KUKA KRL program: MyProgram_066().src

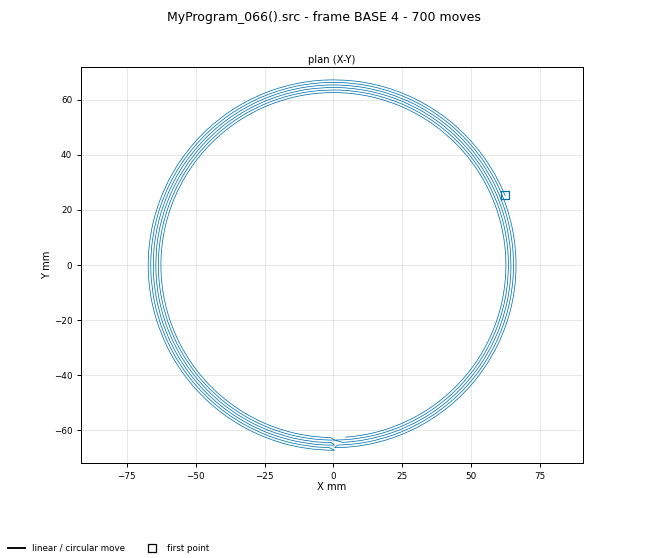
[picture p0: tool path of MyProgram_066().src in frame BASE 4, 700 of 700 moves have a stored position in this frame; points joined in program order, loops and branches not executed]
&ACCESS RVP
&REL 1
&PARAM TEMPLATE = C:\KRC\Roboter\Template\vorgabe
&PARAM EDITMASK = *
DEF MyProgram_066()
; ---- Setting reference (Base) ----
$BASE = BASE_DATA[4]

; --------------------------
; ---- Setting tool (TCP) ----
$TOOL = TOOL_DATA[3]
; --------------------------

$VEL.CP = VEL_APROX_PRINT
Startdeposition()
$VEL.CP = VEL_PRINT
LIN {X 62.3315,Y 25.2881,Z 74,A 16.8534,B 24.8789,C -2.5402,E1 25.1473,E2 67.2399} C_DIS
LIN {X 60.7324,Y 28.9196,Z 74,A 20.0242,B 24.8785,C -2.5441,E1 25.1436,E2 64.0772} C_DIS
LIN {X 58.523,Y 33.1652,Z 74,A 24.2572,B 24.877,C -2.5592,E1 25.138,E2 59.8308} C_DIS
LIN {X 56.2659,Y 36.8633,Z 74,A 27.5694,B 24.877,C -2.5587,E1 25.1331,E2 56.5365} C_DIS
LIN {X 55.2782,Y 38.328,Z 74,A 29.4981,B 24.8757,C -2.5736,E1 25.13,E2 54.5819} C_DIS
LIN {X 52.9232,Y 41.5199,Z 74,A 32.7172,B 24.8753,C -2.5775,E1 25.1246,E2 51.369} C_DIS
LIN {X 49.6306,Y 45.404,Z 74,A 36.4526,B 24.8758,C -2.5716,E1 25.1179,E2 47.6643} C_DIS
LIN {X 47.2788,Y 47.848,Z 74,A 39.6344,B 24.8745,C -2.5853,E1 25.1116,E2 44.4638} C_DIS
LIN {X 44.4374,Y 50.4985,Z 74,A 42.7954,B 24.8742,C -2.5881,E1 25.1051,E2 41.309} C_DIS
LIN {X 41.8737,Y 52.6437,Z 74,A 45.7271,B 24.8735,C -2.5955,E1 25.0988,E2 38.371} C_DIS
LIN {X 38.9575,Y 54.8366,Z 74,A 49.1887,B 24.8721,C -2.6099,E1 25.091,E2 34.8877} C_DIS
LIN {X 35.2683,Y 57.2802,Z 74,A 52.5369,B 24.8726,C -2.6051,E1 25.0832,E2 31.5619} C_DIS
LIN {X 32.0783,Y 59.1244,Z 74,A 55.3853,B 24.8729,C -2.6022,E1 25.0763,E2 28.7288} C_DIS
LIN {X 29.6751,Y 60.3668,Z 74,A 58.2734,B 24.8712,C -2.6196,E1 25.0691,E2 25.8073} C_DIS
LIN {X 27.6413,Y 61.3243,Z 74,A 60.3296,B 24.8706,C -2.6253,E1 25.0638,E2 23.7428} C_DIS
LIN {X 24.27,Y 62.736,Z 74,A 63.3703,B 24.8705,C -2.6266,E1 25.0559,E2 20.7059} C_DIS
LIN {X 20.9505,Y 63.9207,Z 74,A 66.4008,B 24.8701,C -2.6298,E1 25.0479,E2 17.6737} C_DIS
LIN {X 17.9241,Y 64.8352,Z 74,A 69.0945,B 24.87,C -2.6317,E1 25.0407,E2 14.9802} C_DIS
LIN {X 13.9191,Y 65.8114,Z 74,A 72.377,B 24.8703,C -2.6279,E1 25.0318,E2 11.7111} C_DIS
LIN {X 10.864,Y 66.3823,Z 74,A 75.0856,B 24.8701,C -2.6304,E1 25.0243,E2 8.9996} C_DIS
LIN {X 7.712,Y 66.8226,Z 74,A 77.9948,B 24.8696,C -2.6357,E1 25.0163,E2 6.0801} C_DIS
LIN {X 4.131,Y 67.1403,Z 74,A 80.6016,B 24.8706,C -2.625,E1 25.0091,E2 3.5} C_DIS
LIN {X -0.3651,Y 67.265,Z 74,A 84.501,B 24.8706,C -2.6261,E1 24.9982,E2 -0.4014} C_DIS
LIN {X -3.8279,Y 67.1571,Z 74,A 88.2033,B 24.8689,C -2.6427,E1 24.9877,E2 -4.1439} C_DIS
LIN {X -7.4514,Y 66.8531,Z 74,A 90.84,B 24.8701,C -2.6303,E1 24.9805,E2 -6.7528} C_DIS
LIN {X -10.4471,Y 66.45,Z 74,A 93.2751,B 24.8706,C -2.6255,E1 24.9738,E2 -9.1784} C_DIS
LIN {X -12.9697,Y 66.0043,Z 74,A 95.4752,B 24.8706,C -2.6242,E1 24.9678,E2 -11.3777} C_DIS
LIN {X -16.4947,Y 65.2128,Z 74,A 99.486,B 24.8689,C -2.6426,E1 24.9567,E2 -15.438} C_DIS
LIN {X -19.9918,Y 64.2265,Z 74,A 101.0557,B 24.8726,C -2.6048,E1 24.9528,E2 -16.9203} C_DIS
LIN {X -23.3556,Y 63.082,Z 74,A 104.7013,B 24.8716,C -2.6149,E1 24.9431,E2 -20.5968} C_DIS
LIN {X -25.7788,Y 62.1314,Z 74,A 107.2724,B 24.8711,C -2.6197,E1 24.9364,E2 -23.1852} C_DIS
LIN {X -29.9946,Y 60.2084,Z 74,A 110.6168,B 24.873,C -2.6004,E1 24.928,E2 -26.492} C_DIS
LIN {X -31.8168,Y 59.2655,Z 74,A 112.8643,B 24.8722,C -2.6085,E1 24.9224,E2 -28.765} C_DIS
LIN {X -35.093,Y 57.3867,Z 74,A 115.6735,B 24.8737,C -2.5939,E1 24.9157,E2 -31.5478} C_DIS
LIN {X -36.6852,Y 56.3816,Z 74,A 117.6551,B 24.8732,C -2.5991,E1 24.911,E2 -33.5482} C_DIS
LIN {X -39.5297,Y 54.426,Z 74,A 120.8352,B 24.8732,C -2.5984,E1 24.9038,E2 -36.7377} C_DIS
LIN {X -43.4881,Y 51.318,Z 74,A 124.3334,B 24.8758,C -2.5723,E1 24.8963,E2 -40.1869} C_DIS
LIN {X -45.912,Y 49.1611,Z 74,A 127.8706,B 24.8748,C -2.5825,E1 24.8889,E2 -43.7626} C_DIS
LIN {X -49.0981,Y 45.9794,Z 74,A 131.8946,B 24.8753,C -2.5773,E1 24.8811,E2 -47.7914} C_DIS
LIN {X -51.4905,Y 43.285,Z 74,A 134.9532,B 24.8761,C -2.5693,E1 24.8755,E2 -50.8448} C_DIS
LIN {X -54.426,Y 39.5297,Z 74,A 138.5981,B 24.878,C -2.5498,E1 24.8694,E2 -54.4606} C_DIS
LIN {X -56.1384,Y 37.0567,Z 74,A 141.0375,B 24.8789,C -2.5402,E1 24.8656,E2 -56.8894} C_DIS
LIN {X -57.3949,Y 35.0794,Z 74,A 143.5728,B 24.8783,C -2.5459,E1 24.8619,E2 -59.4512} C_DIS
LIN {X -59.9905,Y 30.4285,Z 74,A 148.1441,B 24.8795,C -2.5336,E1 24.8559,E2 -64.0172} C_DIS
LIN {X -62.1829,Y 25.6534,Z 74,A 152.2818,B 24.8814,C -2.5132,E1 24.8512,E2 -68.129} C_DIS
LIN {X -63.6586,Y 21.734,Z 74,A 155.9508,B 24.8823,C -2.5044,E1 24.8477,E2 -71.7979} C_DIS
LIN {X -64.7804,Y 18.1175,Z 74,A 159.2016,B 24.8832,C -2.495,E1 24.8452,E2 -75.0449} C_DIS
LIN {X -65.5151,Y 15.2482,Z 74,A 161.5576,B 24.8842,C -2.4837,E1 24.8436,E2 -77.3876} C_DIS
LIN {X -65.9957,Y 13.0146,Z 74,A 163.4166,B 24.885,C -2.4758,E1 24.8426,E2 -79.2387} C_DIS
LIN {X -66.7571,Y 8.2673,Z 74,A 167.478,B 24.8862,C -2.4621,E1 24.8409,E2 -83.2917} C_DIS
LIN {X -67.1045,Y 4.6607,Z 74,A 171.2927,B 24.8857,C -2.4673,E1 24.84,E2 -87.1417} C_DIS
LIN {X -67.2573,Y 1.0908,Z 74,A 174.6764,B 24.886,C -2.4648,E1 24.8398,E2 -90.5396} C_DIS
LIN {X -67.2266,Y -2.3165,Z 74,A 176.844,B 24.8882,C -2.4404,E1 24.84,E2 -92.662} C_DIS
LIN {X -67.0976,Y -4.7627,Z 74,A 179.1127,B 24.8885,C -2.4376,E1 24.8404,E2 -94.9376} C_DIS
LIN {X -66.7559,Y -8.277,Z 74,A -177.9869,B 24.8895,C -2.426,E1 24.8413,E2 -97.8276} C_DIS
LIN {X -66.2127,Y -11.8575,Z 74,A -174.9721,B 24.8905,C -2.415,E1 24.8426,E2 -100.8342} C_DIS
LIN {X -65.7862,Y -14.0352,Z 74,A -172.2602,B 24.8895,C -2.4264,E1 24.8442,E2 -103.5892} C_DIS
LIN {X -65.0081,Y -17.2788,Z 74,A -170.101,B 24.8916,C -2.4036,E1 24.8457,E2 -105.7065} C_DIS
LIN {X -64.2056,Y -20.0594,Z 74,A -167.7944,B 24.8925,C -2.3929,E1 24.8476,E2 -108.001} C_DIS
LIN {X -63.5273,Y -22.114,Z 74,A -165.4328,B 24.8921,C -2.3984,E1 24.8497,E2 -110.3891} C_DIS
LIN {X -61.4519,Y -27.3582,Z 74,A -161.3561,B 24.8946,C -2.3695,E1 24.854,E2 -114.4193} C_DIS
LIN {X -60.244,Y -29.923,Z 74,A -158.4157,B 24.8943,C -2.3738,E1 24.8576,E2 -117.3862} C_DIS
LIN {X -58.7607,Y -32.7395,Z 74,A -155.6768,B 24.8949,C -2.3672,E1 24.8613,E2 -120.1237} C_DIS
LIN {X -57.5024,Y -34.9027,Z 74,A -153.0961,B 24.8945,C -2.3712,E1 24.865,E2 -122.7273} C_DIS
LIN {X -55.1447,Y -38.5202,Z 74,A -150.0261,B 24.8965,C -2.349,E1 24.8698,E2 -125.7595} C_DIS
LIN {X -53.5092,Y -40.763,Z 74,A -147.4333,B 24.8965,C -2.3482,E1 24.8741,E2 -128.3628} C_DIS
LIN {X -51.3233,Y -43.4818,Z 74,A -144.7496,B 24.8977,C -2.3352,E1 24.8789,E2 -131.0278} C_DIS
LIN {X -49.4277,Y -45.6252,Z 74,A -142.4389,B 24.8984,C -2.3271,E1 24.8832,E2 -133.3295} C_DIS
LIN {X -47.0995,Y -48.0251,Z 74,A -139.4796,B 24.8987,C -2.3235,E1 24.889,E2 -136.293} C_DIS
LIN {X -45.2438,Y -49.7777,Z 74,A -137.0243,B 24.8985,C -2.3253,E1 24.894,E2 -138.7626} C_DIS
LIN {X -43.3659,Y -51.4221,Z 74,A -134.2375,B 24.8976,C -2.336,E1 24.9001,E2 -141.5856} C_DIS
LIN {X -40.7193,Y -53.5426,Z 74,A -131.2988,B 24.898,C -2.3321,E1 24.9066,E2 -144.5256} C_DIS
LIN {X -37.9226,Y -55.5577,Z 74,A -129.4698,B 24.9005,C -2.3026,E1 24.9107,E2 -146.2904} C_DIS
LIN {X -34.8215,Y -57.5517,Z 74,A -125.8623,B 24.9,C -2.3083,E1 24.9192,E2 -149.923} C_DIS
LIN {X -31.8372,Y -59.2552,Z 74,A -123.1085,B 24.9007,C -2.3005,E1 24.9259,E2 -152.6661} C_DIS
LIN {X -29.2171,Y -60.5895,Z 74,A -120.3691,B 24.9005,C -2.3028,E1 24.9328,E2 -155.4183} C_DIS
LIN {X -25.5883,Y -62.2094,Z 74,A -117.097,B 24.901,C -2.2967,E1 24.9412,E2 -158.6834} C_DIS
LIN {X -21.9524,Y -63.5838,Z 74,A -113.698,B 24.9011,C -2.2959,E1 24.9501,E2 -162.0873} C_DIS
LIN {X -18.3294,Y -64.7205,Z 74,A -110.5135,B 24.9014,C -2.2925,E1 24.9586,E2 -165.2691} C_DIS
LIN {X -16.0949,Y -65.3123,Z 74,A -107.5998,B 24.8995,C -2.3138,E1 24.9667,E2 -168.2377} C_DIS
LIN {X -12.1273,Y -66.1641,Z 74,A -103.8828,B 24.8991,C -2.3189,E1 24.977,E2 -171.9705} C_DIS
LIN {X -7.472,Y -66.8507,Z 74,A -100.7261,B 24.901,C -2.2977,E1 24.9856,E2 -175.0788} C_DIS
LIN {X -2.0633,Y -67.2344,Z 74,A -96.425,B 24.9016,C -2.2902,E1 24.9975,E2 -179.3634} C_DIS
LIN {X 0.449,Y -67.2547,Z 74,A -94.5441,B 24.9021,C -2.2846,E1 25.0027,E2 -181.2309} C_DIS
Enddeposition()
LIN {X 0.449,Y -67.2547,Z 74,A -94.5441,B 24.9021,C -2.2846,E1 25.0027,E2 -181.2309} C_DIS
Startdeposition()
$VEL.CP = VEL_PRINT
LIN {X -1.4149,Y -66.3279,Z 74,A -97.2166,B 24.9029,C -2.2748,E1 24.9952,E2 -178.5352} C_DIS
LIN {X -6.4726,Y -66.0273,Z 74,A -101.5733,B 24.9029,C -2.2752,E1 24.9831,E2 -174.1777} C_DIS
LIN {X -11.6127,Y -65.3185,Z 74,A -105.8847,B 24.9025,C -2.2802,E1 24.9712,E2 -169.8746} C_DIS
LIN {X -14.9653,Y -64.6327,Z 74,A -108.7487,B 24.9022,C -2.2835,E1 24.9634,E2 -167.015} C_DIS
LIN {X -17.1256,Y -64.0944,Z 74,A -111.8991,B 24.9044,C -2.2571,E1 24.9547,E2 -163.7972} C_DIS
LIN {X -20.6683,Y -63.0415,Z 74,A -114.2557,B 24.9026,C -2.278,E1 24.9486,E2 -161.486} C_DIS
LIN {X -22.9852,Y -62.2343,Z 74,A -116.4421,B 24.9026,C -2.2783,E1 24.9428,E2 -159.296} C_DIS
LIN {X -25.3695,Y -61.3016,Z 74,A -118.9919,B 24.9031,C -2.2731,E1 24.9362,E2 -156.728} C_DIS
LIN {X -30.5306,Y -58.9014,Z 74,A -123.945,B 24.9026,C -2.2781,E1 24.9237,E2 -151.774} C_DIS
LIN {X -34.4147,Y -56.7185,Z 74,A -127.7165,B 24.902,C -2.2852,E1 24.9147,E2 -148.008} C_DIS
LIN {X -37.3127,Y -54.8555,Z 74,A -130.8798,B 24.902,C -2.2859,E1 24.9073,E2 -144.8358} C_DIS
LIN {X -40.1239,Y -52.835,Z 74,A -133.2241,B 24.9003,C -2.3047,E1 24.9021,E2 -142.528} C_DIS
LIN {X -42.9208,Y -50.5883,Z 74,A -136.3928,B 24.9,C -2.3089,E1 24.8953,E2 -139.3573} C_DIS
LIN {X -45.6353,Y -48.1543,Z 74,A -139.6748,B 24.8997,C -2.3123,E1 24.8885,E2 -136.0701} C_DIS
LIN {X -48.3948,Y -45.3796,Z 74,A -143.0463,B 24.899,C -2.3196,E1 24.882,E2 -132.7017} C_DIS
LIN {X -50.6642,Y -42.8317,Z 74,A -146.3244,B 24.899,C -2.3194,E1 24.876,E2 -129.4082} C_DIS
LIN {X -52.8948,Y -40.0444,Z 74,A -148.636,B 24.897,C -2.3426,E1 24.8721,E2 -127.1409} C_DIS
LIN {X -54.1488,Y -38.3318,Z 74,A -151.1998,B 24.898,C -2.332,E1 24.8678,E2 -124.5394} C_DIS
LIN {X -56.7395,Y -34.38,Z 74,A -154.6858,B 24.896,C -2.3546,E1 24.8626,E2 -121.0896} C_DIS
LIN {X -57.9531,Y -32.2924,Z 74,A -156.8887,B 24.8957,C -2.3577,E1 24.8596,E2 -118.8827} C_DIS
LIN {X -59.2868,Y -29.7714,Z 74,A -159.8608,B 24.896,C -2.3541,E1 24.8557,E2 -115.8861} C_DIS
LIN {X -61.0479,Y -25.9716,Z 74,A -163.5382,B 24.8952,C -2.363,E1 24.8516,E2 -112.2098} C_DIS
LIN {X -62.6169,Y -21.9197,Z 74,A -167.4766,B 24.8946,C -2.3702,E1 24.8478,E2 -108.2663} C_DIS
LIN {X -64.2281,Y -16.6168,Z 74,A -172.1789,B 24.8932,C -2.3862,E1 24.8442,E2 -103.5749} C_DIS
LIN {X -64.8986,Y -13.7717,Z 74,A -174.371,B 24.8919,C -2.4004,E1 24.8429,E2 -101.4039} C_DIS
LIN {X -65.4441,Y -10.8822,Z 74,A -177.4683,B 24.8922,C -2.3972,E1 24.8414,E2 -98.2807} C_DIS
LIN {X -66.1466,Y -5.0997,Z 74,A 178.2949,B 24.8893,C -2.4286,E1 24.8402,E2 -94.0934} C_DIS
LIN {X -66.2816,Y -2.8454,Z 74,A 176.1064,B 24.8892,C -2.43,E1 24.8399,E2 -91.8952} C_DIS
LIN {X -66.3414,Y 0.3365,Z 74,A 173.5212,B 24.8881,C -2.4419,E1 24.8398,E2 -89.3229} C_DIS
LIN {X -66.3053,Y 2.2349,Z 74,A 171.3771,B 24.8885,C -2.4372,E1 24.84,E2 -87.1546} C_DIS
LIN {X -66.0051,Y 6.6877,Z 74,A 167.8104,B 24.8869,C -2.455,E1 24.8408,E2 -83.6091} C_DIS
LIN {X -65.6576,Y 9.5109,Z 74,A 164.9106,B 24.8869,C -2.4541,E1 24.8419,E2 -80.6897} C_DIS
LIN {X -65.0311,Y 13.1272,Z 74,A 162.0301,B 24.8855,C -2.4698,E1 24.8434,E2 -77.8296} C_DIS
LIN {X -64.3433,Y 16.1686,Z 74,A 159.3509,B 24.8847,C -2.4784,E1 24.8451,E2 -75.1554} C_DIS
LIN {X -63.4775,Y 19.2866,Z 74,A 156.7155,B 24.8836,C -2.4902,E1 24.8471,E2 -72.5329} C_DIS
LIN {X -62.1556,Y 23.1965,Z 74,A 152.8909,B 24.8831,C -2.496,E1 24.8507,E2 -68.7003} C_DIS
LIN {X -60.5332,Y 27.1485,Z 74,A 148.6944,B 24.883,C -2.497,E1 24.8553,E2 -64.4832} C_DIS
LIN {X -58.8514,Y 30.625,Z 74,A 145.5471,B 24.8817,C -2.5104,E1 24.8593,E2 -61.351} C_DIS
LIN {X -56.7052,Y 34.4365,Z 74,A 142.0487,B 24.8802,C -2.5267,E1 24.8641,E2 -57.8732} C_DIS
LIN {X -54.8734,Y 37.2862,Z 74,A 139.3938,B 24.8789,C -2.5401,E1 24.8682,E2 -55.2372} C_DIS
LIN {X -53.7459,Y 38.8956,Z 74,A 137.4149,B 24.8789,C -2.539,E1 24.8714,E2 -53.246} C_DIS
LIN {X -51.8231,Y 41.4228,Z 74,A 134.5691,B 24.8785,C -2.5441,E1 24.8763,E2 -50.3989} C_DIS
LIN {X -49.4365,Y 44.2423,Z 74,A 131.2964,B 24.8779,C -2.5505,E1 24.8823,E2 -47.1266} C_DIS
LIN {X -46.9076,Y 46.9168,Z 74,A 128.1251,B 24.8771,C -2.5583,E1 24.8885,E2 -43.9602} C_DIS
LIN {X -44.1214,Y 49.5442,Z 74,A 125.2179,B 24.8756,C -2.5741,E1 24.8944,E2 -41.0789} C_DIS
LIN {X -41.71,Y 51.5909,Z 74,A 122.0987,B 24.8758,C -2.572,E1 24.9011,E2 -37.9429} C_DIS
LIN {X -38.912,Y 53.7338,Z 74,A 119.2437,B 24.8748,C -2.5821,E1 24.9075,E2 -35.1018} C_DIS
LIN {X -36.9584,Y 55.0946,Z 74,A 117.076,B 24.8747,C -2.5838,E1 24.9125,E2 -32.9309} C_DIS
LIN {X -34.4679,Y 56.6861,Z 74,A 114.2062,B 24.8748,C -2.5819,E1 24.9193,E2 -30.0475} C_DIS
LIN {X -30.1508,Y 59.0955,Z 74,A 110.3017,B 24.8734,C -2.5967,E1 24.9288,E2 -26.1673} C_DIS
LIN {X -27.0922,Y 60.559,Z 74,A 106.9855,B 24.8738,C -2.5929,E1 24.9373,E2 -22.8338} C_DIS
LIN {X -23.5832,Y 62.0096,Z 74,A 103.7025,B 24.8734,C -2.5972,E1 24.9458,E2 -19.5539} C_DIS
LIN {X -20.5647,Y 63.0751,Z 74,A 101.4564,B 24.8719,C -2.6117,E1 24.9517,E2 -17.3381} C_DIS
LIN {X -16.4891,Y 64.2609,Z 74,A 97.9439,B 24.8712,C -2.6189,E1 24.9611,E2 -13.8371} C_DIS
LIN {X -13.3428,Y 64.9871,Z 74,A 95.0047,B 24.8713,C -2.6181,E1 24.9691,E2 -10.8921} C_DIS
LIN {X -11.5671,Y 65.3268,Z 74,A 93.1162,B 24.8719,C -2.612,E1 24.9743,E2 -8.9872} C_DIS
LIN {X -7.9595,Y 65.8639,Z 74,A 90.3042,B 24.871,C -2.6215,E1 24.982,E2 -6.1956} C_DIS
LIN {X -4.1713,Y 66.2121,Z 74,A 86.3277,B 24.8723,C -2.6075,E1 24.9932,E2 -2.1841} C_DIS
LIN {X -0.5098,Y 66.3408,Z 74,A 82.8327,B 24.873,C -2.6009,E1 25.003,E2 1.3268} C_DIS
LIN {X 2.8294,Y 66.2823,Z 74,A 81.3016,B 24.8699,C -2.6319,E1 25.0071,E2 2.7839} C_DIS
LIN {X 4.7605,Y 66.1723,Z 74,A 78.5897,B 24.8723,C -2.608,E1 25.0148,E2 5.5513} C_DIS
LIN {X 9.6031,Y 65.6446,Z 74,A 74.5516,B 24.872,C -2.611,E1 25.0259,E2 9.5791} C_DIS
LIN {X 12.7089,Y 65.1142,Z 74,A 72.1013,B 24.8715,C -2.6162,E1 25.0326,E2 12.0142} C_DIS
LIN {X 16.0999,Y 64.3597,Z 74,A 69.1183,B 24.8716,C -2.6151,E1 25.0407,E2 14.9958} C_DIS
LIN {X 20.0962,Y 63.2267,Z 74,A 65.8599,B 24.8711,C -2.6203,E1 25.0494,E2 18.2362} C_DIS
LIN {X 24.5864,Y 61.6194,Z 74,A 61.0061,B 24.8732,C -2.5991,E1 25.0622,E2 23.1301} C_DIS
LIN {X 27.6395,Y 60.3122,Z 74,A 58.4966,B 24.8726,C -2.6045,E1 25.0686,E2 25.6207} C_DIS
LIN {X 31.5817,Y 58.3434,Z 74,A 54.322,B 24.874,C -2.5907,E1 25.079,E2 29.8162} C_DIS
LIN {X 34.8131,Y 56.4761,Z 74,A 50.7144,B 24.8754,C -2.5767,E1 25.0876,E2 33.4458} C_DIS
LIN {X 37.7449,Y 54.5591,Z 74,A 47.7125,B 24.8758,C -2.5723,E1 25.0945,E2 36.4478} C_DIS
LIN {X 40.5739,Y 52.4893,Z 74,A 46.1787,B 24.8727,C -2.6038,E1 25.0978,E2 37.9015} C_DIS
LIN {X 42.6402,Y 50.8257,Z 74,A 43.3374,B 24.8745,C -2.5859,E1 25.104,E2 40.7745} C_DIS
LIN {X 44.2021,Y 49.4725,Z 74,A 41.099,B 24.8759,C -2.5711,E1 25.1087,E2 43.0389} C_DIS
LIN {X 46.5542,Y 47.2659,Z 74,A 38.3066,B 24.8765,C -2.5652,E1 25.1143,E2 45.8337} C_DIS
LIN {X 48.7959,Y 44.9481,Z 74,A 36.1102,B 24.8756,C -2.5739,E1 25.1185,E2 47.9998} C_DIS
LIN {X 51.1276,Y 42.2771,Z 74,A 32.8841,B 24.8767,C -2.5628,E1 25.1244,E2 51.2377} C_DIS
LIN {X 53.4624,Y 39.2827,Z 74,A 29.9082,B 24.8767,C -2.5627,E1 25.1294,E2 54.1996} C_DIS
LIN {X 54.7371,Y 37.4876,Z 74,A 27.6827,B 24.878,C -2.5497,E1 25.133,E2 56.445} C_DIS
LIN {X 57.5072,Y 33.0798,Z 74,A 23.595,B 24.878,C -2.5486,E1 25.139,E2 60.5147} C_DIS
LIN {X 59.3392,Y 29.6693,Z 74,A 20.1707,B 24.8791,C -2.5374,E1 25.1434,E2 63.9472} C_DIS
LIN {X 60.8589,Y 26.4102,Z 74,A 16.1566,B 24.8822,C -2.5053,E1 25.1481,E2 68.0154} C_DIS
LIN {X 62.4219,Y 22.4707,Z 74,A 12.8782,B 24.8822,C -2.5045,E1 25.1513,E2 71.2773} C_DIS
LIN {X 63.5424,Y 19.0726,Z 74,A 9.9293,B 24.8828,C -2.4991,E1 25.1537,E2 74.2224} C_DIS
LIN {X 64.6929,Y 14.705,Z 74,A 6.7032,B 24.8822,C -2.5049,E1 25.1559,E2 77.416} C_DIS
LIN {X 65.4196,Y 11.0285,Z 74,A 3.1661,B 24.8839,C -2.4871,E1 25.1578,E2 80.9747} C_DIS
LIN {X 65.9012,Y 7.6411,Z 74,A -0.297,B 24.886,C -2.4646,E1 25.159,E2 84.4705} C_DIS
LIN {X 66.3011,Y 2.3596,Z 74,A -5.0224,B 24.8877,C -2.4462,E1 25.1598,E2 89.2111} C_DIS
LIN {X 66.3122,Y -2.0111,Z 74,A -8.7803,B 24.8887,C -2.4347,E1 25.1596,E2 92.9739} C_DIS
LIN {X 66.1167,Y -5.4741,Z 74,A -11.2155,B 24.8883,C -2.4399,E1 25.1591,E2 95.3824} C_DIS
LIN {X 65.8624,Y -7.9729,Z 74,A -14.1349,B 24.8907,C -2.4134,E1 25.1581,E2 98.3473} C_DIS
LIN {X 65.3481,Y -11.4482,Z 74,A -16.3481,B 24.8896,C -2.4252,E1 25.1571,E2 100.5194} C_DIS
LIN {X 64.6009,Y -15.103,Z 74,A -19.0559,B 24.8893,C -2.4287,E1 25.1555,E2 103.2033} C_DIS
LIN {X 63.9973,Y -17.485,Z 74,A -21.728,B 24.8912,C -2.4075,E1 25.1536,E2 105.91} C_DIS
LIN {X 62.9902,Y -20.8263,Z 74,A -24.4104,B 24.8912,C -2.4069,E1 25.1514,E2 108.5786} C_DIS
LIN {X 62.405,Y -22.517,Z 74,A -26.3509,B 24.8926,C -2.3918,E1 25.1495,E2 110.5438} C_DIS
LIN {X 61.0444,Y -25.9805,Z 74,A -29.3909,B 24.8931,C -2.3867,E1 25.1463,E2 113.5793} C_DIS
LIN {X 59.7124,Y -28.9106,Z 74,A -31.9702,B 24.8934,C -2.3837,E1 25.1433,E2 116.1516} C_DIS
LIN {X 58.693,Y -30.927,Z 74,A -34.428,B 24.8951,C -2.3648,E1 25.1401,E2 118.641} C_DIS
LIN {X 56.0131,Y -35.5528,Z 74,A -39.3479,B 24.8969,C -2.344,E1 25.1329,E2 123.5852} C_DIS
LIN {X 52.8789,Y -40.0655,Z 74,A -43.4784,B 24.8966,C -2.347,E1 25.1262,E2 127.6885} C_DIS
LIN {X 50.4209,Y -43.1173,Z 74,A -46.5566,B 24.8967,C -2.3462,E1 25.1208,E2 130.7545} C_DIS
LIN {X 48.7061,Y -45.0459,Z 74,A -49.3264,B 24.8984,C -2.3267,E1 25.1155,E2 133.558} C_DIS
LIN {X 45.8322,Y -47.9671,Z 74,A -52.5835,B 24.8985,C -2.3255,E1 25.109,E2 136.8045} C_DIS
LIN {X 42.9448,Y -50.5678,Z 74,A -55.619,B 24.8985,C -2.3261,E1 25.1027,E2 139.8264} C_DIS
LIN {X 40.8106,Y -52.3068,Z 74,A -58.6063,B 24.9003,C -2.3055,E1 25.0961,E2 142.8513} C_DIS
LIN {X 37.5193,Y -54.7157,Z 74,A -61.9311,B 24.9005,C -2.3034,E1 25.0885,E2 146.1696} C_DIS
LIN {X 33.7271,Y -57.13,Z 74,A -65.3568,B 24.9001,C -2.3076,E1 25.0805,E2 149.5743} C_DIS
LIN {X 30.4588,Y -58.9381,Z 74,A -69.1225,B 24.9017,C -2.2887,E1 25.0711,E2 153.3741} C_DIS
LIN {X 27.4535,Y -60.3962,Z 74,A -71.4428,B 24.9009,C -2.2982,E1 25.0653,E2 155.6661} C_DIS
LIN {X 24.8438,Y -61.5156,Z 74,A -74.1691,B 24.9018,C -2.2879,E1 25.0582,E2 158.4103} C_DIS
LIN {X 21.7194,Y -62.6872,Z 74,A -77.0242,B 24.9021,C -2.2848,E1 25.0507,E2 161.2668} C_DIS
LIN {X 19.056,Y -63.5473,Z 74,A -79.2329,B 24.9019,C -2.2871,E1 25.0449,E2 163.4661} C_DIS
LIN {X 15.7348,Y -64.4497,Z 74,A -82.1503,B 24.902,C -2.2854,E1 25.037,E2 166.383} C_DIS
LIN {X 13.1909,Y -65.0183,Z 74,A -85.667,B 24.9048,C -2.2532,E1 25.0272,E2 169.9716} C_DIS
LIN {X 9.0782,Y -65.7191,Z 74,A -88.0993,B 24.9026,C -2.2784,E1 25.0206,E2 172.3419} C_DIS
LIN {X 4.5562,Y -66.1861,Z 74,A -91.975,B 24.9026,C -2.2776,E1 25.0099,E2 176.2173} C_DIS
LIN {X 0.436,Y -66.3027,Z 74,A -94.6637,B 24.9009,C -2.2977,E1 25.0025,E2 178.8575} C_DIS
Enddeposition()
LIN {X 0.436,Y -66.3027,Z 74,A -94.6637,B 24.9009,C -2.2977,E1 25.0025,E2 178.8575} C_DIS
Startdeposition()
$VEL.CP = VEL_PRINT
LIN {X 1.5364,Y -65.4021,Z 74,A -92.9082,B 24.898,C -2.332,E1 25.0076,E2 177.021} C_DIS
LIN {X 6.6679,Y -65.0788,Z 74,A -88.8013,B 24.8986,C -2.3247,E1 25.019,E2 172.9336} C_DIS
LIN {X 9.6588,Y -64.7026,Z 74,A -85.5651,B 24.8972,C -2.3409,E1 25.028,E2 169.6618} C_DIS
LIN {X 13.0107,Y -64.1127,Z 74,A -83.4329,B 24.8988,C -2.3227,E1 25.0338,E2 167.5753} C_DIS
LIN {X 15.2589,Y -63.6154,Z 74,A -81.1168,B 24.898,C -2.3319,E1 25.0401,E2 165.2406} C_DIS
LIN {X 18.93,Y -62.6209,Z 74,A -78.0568,B 24.8982,C -2.3289,E1 25.0483,E2 162.1929} C_DIS
LIN {X 21.4935,Y -61.7879,Z 74,A -75.8242,B 24.8982,C -2.3287,E1 25.0542,E2 159.9653} C_DIS
LIN {X 24.6283,Y -60.6064,Z 74,A -72.403,B 24.8968,C -2.3448,E1 25.0631,E2 156.5135} C_DIS
LIN {X 27.6955,Y -59.2677,Z 74,A -69.3685,B 24.8962,C -2.3519,E1 25.0709,E2 153.4699} C_DIS
LIN {X 32.5774,Y -56.731,Z 74,A -65.2367,B 24.897,C -2.3428,E1 25.0809,E2 149.3714} C_DIS
LIN {X 37.0028,Y -53.9503,Z 74,A -60.1787,B 24.8952,C -2.3636,E1 25.0929,E2 144.2806} C_DIS
LIN {X 40.9187,Y -51.0438,Z 74,A -56.3828,B 24.8955,C -2.3604,E1 25.1013,E2 140.506} C_DIS
LIN {X 43.7208,Y -48.6627,Z 74,A -52.8437,B 24.8941,C -2.3759,E1 25.1088,E2 136.9443} C_DIS
LIN {X 46.6882,Y -45.8246,Z 74,A -48.9761,B 24.8927,C -2.3915,E1 25.1165,E2 133.0561} C_DIS
LIN {X 49.3002,Y -43.0021,Z 74,A -45.7073,B 24.8921,C -2.3974,E1 25.1225,E2 129.788} C_DIS
LIN {X 52.2689,Y -39.3403,Z 74,A -42.2274,B 24.8927,C -2.3913,E1 25.1285,E2 126.3388} C_DIS
LIN {X 54.8518,Y -35.6526,Z 74,A -38.1206,B 24.8913,C -2.4063,E1 25.135,E2 122.2167} C_DIS
LIN {X 56.3517,Y -33.2292,Z 74,A -35.5259,B 24.8905,C -2.416,E1 25.1388,E2 119.6124} C_DIS
LIN {X 57.9792,Y -30.3009,Z 74,A -32.7385,B 24.89,C -2.4206,E1 25.1425,E2 116.8287} C_DIS
LIN {X 59.5125,Y -27.167,Z 74,A -29.4159,B 24.8886,C -2.4366,E1 25.1464,E2 113.4861} C_DIS
LIN {X 60.8339,Y -24.0614,Z 74,A -26.7442,B 24.8884,C -2.4381,E1 25.1493,E2 110.8258} C_DIS
LIN {X 61.7874,Y -21.4951,Z 74,A -24.3517,B 24.8878,C -2.4452,E1 25.1515,E2 108.4297} C_DIS
LIN {X 62.6656,Y -18.7809,Z 74,A -21.1293,B 24.8853,C -2.4722,E1 25.1542,E2 105.1619} C_DIS
LIN {X 63.5166,Y -15.6641,Z 74,A -19.0424,B 24.8863,C -2.4613,E1 25.1556,E2 103.1129} C_DIS
LIN {X 64.4274,Y -11.3513,Z 74,A -15.1224,B 24.885,C -2.475,E1 25.1577,E2 99.1834} C_DIS
LIN {X 65.0317,Y -7.118,Z 74,A -11.6132,B 24.8845,C -2.4806,E1 25.159,E2 95.6816} C_DIS
LIN {X 65.3209,Y -3.5886,Z 74,A -7.8934,B 24.882,C -2.5069,E1 25.1597,E2 91.9219} C_DIS
LIN {X 65.4157,Y 0.6341,Z 74,A -3.7748,B 24.8799,C -2.5298,E1 25.1597,E2 87.7736} C_DIS
LIN {X 65.2677,Y 4.4515,Z 74,A -1.4271,B 24.8814,C -2.5137,E1 25.1593,E2 85.4778} C_DIS
LIN {X 64.9167,Y 8.0894,Z 74,A 1.8323,B 24.8803,C -2.5253,E1 25.1583,E2 82.2104} C_DIS
LIN {X 64.437,Y 11.2895,Z 74,A 4.8588,B 24.879,C -2.5391,E1 25.1569,E2 79.169} C_DIS
LIN {X 63.6506,Y 15.1148,Z 74,A 8.3925,B 24.8777,C -2.5525,E1 25.1547,E2 75.6242} C_DIS
LIN {X 62.6049,Y 18.9862,Z 74,A 11.4038,B 24.878,C -2.5498,E1 25.1524,E2 72.6365} C_DIS
LIN {X 61.6622,Y 21.8518,Z 74,A 14.1234,B 24.877,C -2.5596,E1 25.15,E2 69.9091} C_DIS
LIN {X 60.2378,Y 25.5168,Z 74,A 17.8439,B 24.8754,C -2.5766,E1 25.1461,E2 66.1688} C_DIS
LIN {X 58.6832,Y 28.9137,Z 74,A 20.7256,B 24.8754,C -2.5755,E1 25.1426,E2 63.3052} C_DIS
LIN {X 57.2804,Y 31.603,Z 74,A 23.4417,B 24.8746,C -2.5842,E1 25.139,E2 60.5829} C_DIS
LIN {X 55.0885,Y 35.2839,Z 74,A 27.099,B 24.8739,C -2.5915,E1 25.1337,E2 56.9269} C_DIS
LIN {X 53.7088,Y 37.3505,Z 74,A 29.5127,B 24.8728,C -2.603,E1 25.1299,E2 54.4978} C_DIS
LIN {X 50.9751,Y 41.0036,Z 74,A 32.9753,B 24.8732,C -2.5989,E1 25.124,E2 51.0614} C_DIS
LIN {X 49.3107,Y 42.9901,Z 74,A 35.6546,B 24.8717,C -2.6145,E1 25.1191,E2 48.3575} C_DIS
LIN {X 47.1892,Y 45.3087,Z 74,A 38.5987,B 24.8706,C -2.6253,E1 25.1135,E2 45.4005} C_DIS
LIN {X 43.9661,Y 48.4436,Z 74,A 42.2066,B 24.8706,C -2.6249,E1 25.1062,E2 41.8084} C_DIS
LIN {X 41.3767,Y 50.6726,Z 74,A 45.2741,B 24.8699,C -2.6324,E1 25.0996,E2 38.7349} C_DIS
LIN {X 38.0329,Y 53.2277,Z 74,A 48.6723,B 24.8699,C -2.6317,E1 25.092,E2 35.3507} C_DIS
LIN {X 36.5719,Y 54.2421,Z 74,A 50.9573,B 24.8679,C -2.6522,E1 25.0866,E2 33.0248} C_DIS
LIN {X 32.888,Y 56.5525,Z 74,A 54.4648,B 24.8681,C -2.6503,E1 25.0783,E2 29.5327} C_DIS
LIN {X 29.5236,Y 58.3789,Z 74,A 57.9082,B 24.8675,C -2.6568,E1 25.0697,E2 26.0834} C_DIS
LIN {X 26.7428,Y 59.7037,Z 74,A 60.7125,B 24.8669,C -2.6624,E1 25.0626,E2 23.2728} C_DIS
LIN {X 22.1867,Y 61.5427,Z 74,A 64.3713,B 24.868,C -2.651,E1 25.0532,E2 19.649} C_DIS
LIN {X 19.5923,Y 62.417,Z 74,A 66.501,B 24.8685,C -2.6466,E1 25.0475,E2 17.5339} C_DIS
LIN {X 17.1939,Y 63.1196,Z 74,A 69.6421,B 24.8661,C -2.6706,E1 25.039,E2 14.341} C_DIS
LIN {X 13.0654,Y 64.1015,Z 74,A 72.8666,B 24.8671,C -2.6608,E1 25.0302,E2 11.1441} C_DIS
LIN {X 10.6194,Y 64.5519,Z 74,A 74.7202,B 24.8677,C -2.654,E1 25.0252,E2 9.3086} C_DIS
LIN {X 8.9451,Y 64.8054,Z 74,A 77.4555,B 24.8648,C -2.6835,E1 25.0174,E2 6.5053} C_DIS
LIN {X 5.1599,Y 65.2156,Z 74,A 79.8458,B 24.867,C -2.6618,E1 25.0109,E2 4.1679} C_DIS
LIN {X 2.0469,Y 65.3873,Z 74,A 82.5884,B 24.867,C -2.662,E1 25.0033,E2 1.4258} C_DIS
LIN {X -1.8924,Y 65.3921,Z 74,A 87.2051,B 24.8643,C -2.6878,E1 24.9902,E2 -3.2527} C_DIS
LIN {X -6.2763,Y 65.1181,Z 74,A 89.8808,B 24.8672,C -2.6594,E1 24.983,E2 -5.862} C_DIS
LIN {X -9.2473,Y 64.7625,Z 74,A 92.7544,B 24.8668,C -2.6634,E1 24.975,E2 -8.7474} C_DIS
LIN {X -12.4284,Y 64.2279,Z 74,A 96.0899,B 24.8659,C -2.6726,E1 24.9658,E2 -12.1085} C_DIS
LIN {X -15.726,Y 63.5014,Z 74,A 97.9844,B 24.8685,C -2.6464,E1 24.9608,E2 -13.9431} C_DIS
LIN {X -17.912,Y 62.9193,Z 74,A 100.0916,B 24.8685,C -2.6471,E1 24.9551,E2 -16.0553} C_DIS
LIN {X -20.9563,Y 61.972,Z 74,A 103.3878,B 24.8677,C -2.6548,E1 24.9463,E2 -19.3759} C_DIS
LIN {X -24.2931,Y 60.7429,Z 74,A 106.2281,B 24.8687,C -2.6448,E1 24.9389,E2 -22.1982} C_DIS
LIN {X -27.472,Y 59.3717,Z 74,A 109.4028,B 24.8687,C -2.6434,E1 24.9308,E2 -25.3773} C_DIS
LIN {X -30.3844,Y 57.9352,Z 74,A 112.3395,B 24.8691,C -2.6408,E1 24.9235,E2 -28.3157} C_DIS
LIN {X -33.8428,Y 55.9856,Z 74,A 115.7406,B 24.8698,C -2.633,E1 24.9153,E2 -31.7086} C_DIS
LIN {X -37.2356,Y 53.7886,Z 74,A 119.0102,B 24.8711,C -2.6206,E1 24.9078,E2 -34.9592} C_DIS
LIN {X -39.8576,Y 51.8752,Z 74,A 122.7614,B 24.8698,C -2.6337,E1 24.8993,E2 -38.7554} C_DIS
LIN {X -42.4675,Y 49.7615,Z 74,A 124.5978,B 24.8727,C -2.6043,E1 24.8955,E2 -40.5286} C_DIS
LIN {X -44.4078,Y 48.0378,Z 74,A 127.1438,B 24.8727,C -2.6048,E1 24.8902,E2 -43.0859} C_DIS
LIN {X -46.2517,Y 46.2669,Z 74,A 129.4194,B 24.8731,C -2.6002,E1 24.8857,E2 -45.3602} C_DIS
LIN {X -47.9541,Y 44.4979,Z 74,A 132.2043,B 24.8723,C -2.6081,E1 24.8803,E2 -48.176} C_DIS
LIN {X -50.2092,Y 41.9375,Z 74,A 135.3376,B 24.8727,C -2.6034,E1 24.8747,E2 -51.3126} C_DIS
LIN {X -53.0651,Y 38.2609,Z 74,A 138.5326,B 24.8756,C -2.5746,E1 24.8694,E2 -54.4542} C_DIS
LIN {X -54.9186,Y 35.5486,Z 74,A 141.8889,B 24.8754,C -2.5764,E1 24.8642,E2 -57.8315} C_DIS
LIN {X -56.8346,Y 32.397,Z 74,A 145.0341,B 24.8764,C -2.5656,E1 24.8598,E2 -60.9671} C_DIS
LIN {X -58.157,Y 29.9582,Z 74,A 147.128,B 24.8778,C -2.5518,E1 24.8571,E2 -63.0392} C_DIS
LIN {X -59.5472,Y 27.0897,Z 74,A 150.5958,B 24.8772,C -2.5571,E1 24.8529,E2 -66.5387} C_DIS
LIN {X -60.941,Y 23.7887,Z 74,A 153.5417,B 24.8785,C -2.5438,E1 24.8499,E2 -69.4692} C_DIS
LIN {X -62.241,Y 20.1431,Z 74,A 156.4602,B 24.8804,C -2.5241,E1 24.8473,E2 -72.3571} C_DIS
LIN {X -62.7601,Y 18.4627,Z 74,A 158.2228,B 24.8804,C -2.5237,E1 24.8458,E2 -74.129} C_DIS
LIN {X -63.4427,Y 15.9632,Z 74,A 160.7064,B 24.8807,C -2.5209,E1 24.8441,E2 -76.6204} C_DIS
LIN {X -64.2659,Y 12.2311,Z 74,A 164.0045,B 24.8818,C -2.5094,E1 24.8422,E2 -79.9105} C_DIS
LIN {X -64.7725,Y 9.1772,Z 74,A 166.6605,B 24.8827,C -2.4998,E1 24.8411,E2 -82.5593} C_DIS
LIN {X -65.1225,Y 6.2285,Z 74,A 169.6064,B 24.8828,C -2.4984,E1 24.8403,E2 -85.5195} C_DIS
LIN {X -65.3757,Y 2.4116,Z 74,A 173.2875,B 24.8832,C -2.4944,E1 24.8398,E2 -89.2132} C_DIS
LIN {X -65.3873,Y -2.0473,Z 74,A 176.5985,B 24.8855,C -2.4702,E1 24.8399,E2 -92.4864} C_DIS
LIN {X -65.1934,Y -5.4376,Z 74,A 179.9559,B 24.8856,C -2.4685,E1 24.8406,E2 -95.8599} C_DIS
LIN {X -64.6364,Y -10.0913,Z 74,A -176.2705,B 24.8874,C -2.4492,E1 24.842,E2 -99.6098} C_DIS
LIN {X -64.0892,Y -13.1252,Z 74,A -173.582,B 24.8882,C -2.4406,E1 24.8434,E2 -102.2937} C_DIS
LIN {X -62.7107,Y -18.6294,Z 74,A -168.504,B 24.8894,C -2.4279,E1 24.847,E2 -107.3708} C_DIS
LIN {X -61.7066,Y -21.7253,Z 74,A -165.2232,B 24.8894,C -2.4282,E1 24.85,E2 -110.6712} C_DIS
LIN {X -59.9263,Y -26.2402,Z 74,A -161.4443,B 24.8913,C -2.4066,E1 24.854,E2 -114.4193} C_DIS
LIN {X -59.0642,Y -28.1277,Z 74,A -158.8422,B 24.8903,C -2.4176,E1 24.8572,E2 -117.0619} C_DIS
LIN {X -57.5984,Y -31.0187,Z 74,A -156.5259,B 24.892,C -2.3992,E1 24.8602,E2 -119.3465} C_DIS
LIN {X -55.9766,Y -33.8574,Z 74,A -153.6209,B 24.8926,C -2.3926,E1 24.8643,E2 -122.2507} C_DIS
LIN {X -53.9571,Y -36.9909,Z 74,A -150.203,B 24.893,C -2.3876,E1 24.8696,E2 -125.6737} C_DIS
LIN {X -52.0057,Y -39.6887,Z 74,A -147.523,B 24.8941,C -2.3756,E1 24.8741,E2 -128.3381} C_DIS
LIN {X -50.0052,Y -42.1815,Z 74,A -144.4374,B 24.8941,C -2.3752,E1 24.8796,E2 -131.437} C_DIS
LIN {X -47.522,Y -44.9598,Z 74,A -141.5939,B 24.8956,C -2.3593,E1 24.8849,E2 -134.255} C_DIS
LIN {X -44.9775,Y -47.5054,Z 74,A -137.7615,B 24.8948,C -2.3673,E1 24.8927,E2 -138.1224} C_DIS
LIN {X -42.1931,Y -49.9953,Z 74,A -135.2324,B 24.8968,C -2.3452,E1 24.898,E2 -140.6087} C_DIS
LIN {X -39.5169,Y -52.1362,Z 74,A -132.1775,B 24.8972,C -2.341,E1 24.9047,E2 -143.6648} C_DIS
LIN {X -36.7029,Y -54.1534,Z 74,A -129.1618,B 24.8976,C -2.3356,E1 24.9116,E2 -146.6783} C_DIS
LIN {X -34.0079,Y -55.8852,Z 74,A -126.0965,B 24.8976,C -2.3371,E1 24.9188,E2 -149.7567} C_DIS
LIN {X -30.618,Y -57.8122,Z 74,A -122.8722,B 24.8983,C -2.3284,E1 24.9267,E2 -152.9694} C_DIS
LIN {X -29.0433,Y -58.6189,Z 74,A -120.875,B 24.8976,C -2.3364,E1 24.9317,E2 -154.991} C_DIS
LIN {X -25.1505,Y -60.3922,Z 74,A -117.5919,B 24.8988,C -2.3221,E1 24.9401,E2 -158.2478} C_DIS
LIN {X -22.5035,Y -61.4271,Z 74,A -115.5135,B 24.8998,C -2.3107,E1 24.9454,E2 -160.3035} C_DIS
LIN {X -19.9785,Y -62.2943,Z 74,A -112.1688,B 24.898,C -2.3314,E1 24.9544,E2 -163.7039} C_DIS
LIN {X -16.0986,Y -63.4079,Z 74,A -109.0823,B 24.8991,C -2.3191,E1 24.9627,E2 -166.7656} C_DIS
LIN {X -13.8192,Y -63.9432,Z 74,A -107.2546,B 24.8996,C -2.313,E1 24.9676,E2 -168.5813} C_DIS
LIN {X -11.0975,Y -64.4718,Z 74,A -103.935,B 24.8979,C -2.3328,E1 24.9769,E2 -171.9512} C_DIS
LIN {X -6.331,Y -65.1131,Z 74,A -100.5763,B 24.8997,C -2.3123,E1 24.9861,E2 -175.2634} C_DIS
LIN {X -2.7033,Y -65.3636,Z 74,A -97.2101,B 24.8993,C -2.3167,E1 24.9955,E2 -178.6411} C_DIS
LIN {X 0.4342,Y -65.4044,Z 74,A -95.3272,B 24.901,C -2.2972,E1 25.0007,E2 -180.4778} C_DIS
Enddeposition()
LIN {X 0.4342,Y -65.4044,Z 74,A -95.3272,B 24.901,C -2.2972,E1 25.0007,E2 -180.4778} C_DIS
Startdeposition()
$VEL.CP = VEL_PRINT
LIN {X -0.7316,Y -64.4927,Z 74,A -96.4518,B 24.8998,C -2.3108,E1 24.9976,E2 -179.3854} C_DIS
LIN {X -4.0596,Y -64.3688,Z 74,A -99.6455,B 24.9003,C -2.3052,E1 24.9886,E2 -176.1778} C_DIS
LIN {X -6.8131,Y -64.1352,Z 74,A -102.1504,B 24.9003,C -2.3043,E1 24.9817,E2 -173.6693} C_DIS
LIN {X -10.5805,Y -63.6223,Z 74,A -105.8042,B 24.9008,C -2.299,E1 24.9715,E2 -169.9998} C_DIS
LIN {X -13.8299,Y -62.9959,Z 74,A -108.3735,B 24.9,C -2.3083,E1 24.9646,E2 -167.4498} C_DIS
LIN {X -16.2387,Y -62.4186,Z 74,A -110.7129,B 24.9002,C -2.3065,E1 24.9582,E2 -165.1027} C_DIS
LIN {X -21.2426,Y -60.8975,Z 74,A -115.0756,B 24.8994,C -2.316,E1 24.9466,E2 -160.755} C_DIS
LIN {X -24.9313,Y -59.4826,Z 74,A -118.7447,B 24.8994,C -2.3159,E1 24.9371,E2 -157.0777} C_DIS
LIN {X -27.3439,Y -58.4129,Z 74,A -121.0862,B 24.8991,C -2.3185,E1 24.9311,E2 -154.7367} C_DIS
LIN {X -29.6958,Y -57.2542,Z 74,A -123.5864,B 24.8992,C -2.3178,E1 24.9249,E2 -152.228} C_DIS
LIN {X -33.6011,Y -55.052,Z 74,A -127.5602,B 24.8987,C -2.3235,E1 24.9153,E2 -148.256} C_DIS
LIN {X -36.093,Y -53.4513,Z 74,A -130.315,B 24.8986,C -2.325,E1 24.9088,E2 -145.4959} C_DIS
LIN {X -38.9099,Y -51.4373,Z 74,A -134.092,B 24.8994,C -2.3159,E1 24.9003,E2 -141.6837} C_DIS
LIN {X -41.5644,Y -49.3179,Z 74,A -136.6626,B 24.8981,C -2.3306,E1 24.8948,E2 -139.1382} C_DIS
LIN {X -44.3197,Y -46.8565,Z 74,A -139.5575,B 24.8968,C -2.3449,E1 24.8889,E2 -136.2658} C_DIS
LIN {X -46.3669,Y -44.8314,Z 74,A -142.195,B 24.8965,C -2.3487,E1 24.8837,E2 -133.626} C_DIS
LIN {X -49.3461,Y -41.5313,Z 74,A -146.5331,B 24.8965,C -2.3497,E1 24.8757,E2 -129.2709} C_DIS
LIN {X -51.2799,Y -39.1179,Z 74,A -148.6716,B 24.8948,C -2.3683,E1 24.8721,E2 -127.1666} C_DIS
LIN {X -53.3256,Y -36.2786,Z 74,A -152.2598,B 24.8949,C -2.3665,E1 24.8663,E2 -123.5564} C_DIS
LIN {X -55.2138,Y -33.3348,Z 74,A -155.0038,B 24.8936,C -2.3816,E1 24.8623,E2 -120.8345} C_DIS
LIN {X -56.7138,Y -30.7129,Z 74,A -158.2821,B 24.894,C -2.3771,E1 24.8578,E2 -117.5283} C_DIS
LIN {X -58.1454,Y -27.9078,Z 74,A -160.677,B 24.8926,C -2.3926,E1 24.8549,E2 -115.1574} C_DIS
LIN {X -59.3494,Y -25.2475,Z 74,A -164.0573,B 24.8933,C -2.3847,E1 24.8511,E2 -111.7397} C_DIS
LIN {X -60.543,Y -22.2316,Z 74,A -166.0459,B 24.891,C -2.4102,E1 24.8492,E2 -109.8008} C_DIS
LIN {X -61.96,Y -17.9112,Z 74,A -171.005,B 24.8915,C -2.4045,E1 24.8451,E2 -104.7996} C_DIS
LIN {X -62.7747,Y -14.804,Z 74,A -173.0794,B 24.8894,C -2.428,E1 24.8437,E2 -102.769} C_DIS
LIN {X -63.3551,Y -12.0781,Z 74,A -175.6087,B 24.8888,C -2.4345,E1 24.8423,E2 -100.2405} C_DIS
LIN {X -63.8231,Y -9.2949,Z 74,A -178.2911,B 24.8884,C -2.4389,E1 24.8412,E2 -97.5527} C_DIS
LIN {X -64.237,Y -5.7765,Z 74,A 179.1271,B 24.8865,C -2.4595,E1 24.8404,E2 -95.0046} C_DIS
LIN {X -64.4491,Y -2.4764,Z 74,A 175.752,B 24.8864,C -2.4604,E1 24.8398,E2 -91.6113} C_DIS
LIN {X -64.4946,Y 0.3536,Z 74,A 172.8777,B 24.8863,C -2.4616,E1 24.8398,E2 -88.7225} C_DIS
LIN {X -64.2807,Y 5.2676,Z 74,A 169.0778,B 24.884,C -2.4862,E1 24.8404,E2 -84.9586} C_DIS
LIN {X -64.0858,Y 7.2668,Z 74,A 167.0779,B 24.8838,C -2.4877,E1 24.841,E2 -82.9504} C_DIS
LIN {X -63.7052,Y 10.0712,Z 74,A 164.4305,B 24.8833,C -2.4932,E1 24.8421,E2 -80.3001} C_DIS
LIN {X -62.9953,Y 13.8323,Z 74,A 160.832,B 24.8827,C -2.5001,E1 24.844,E2 -76.6969} C_DIS
LIN {X -62.3056,Y 16.6666,Z 74,A 158.6083,B 24.8813,C -2.5151,E1 24.8456,E2 -74.4962} C_DIS
LIN {X -61.3373,Y 19.937,Z 74,A 155.1702,B 24.8811,C -2.5167,E1 24.8484,E2 -71.0421} C_DIS
LIN {X -60.3825,Y 22.6655,Z 74,A 152.7783,B 24.88,C -2.5278,E1 24.8507,E2 -68.6633} C_DIS
LIN {X -58.831,Y 26.4318,Z 74,A 149.3122,B 24.8787,C -2.5416,E1 24.8544,E2 -65.2108} C_DIS
LIN {X -57.8761,Y 28.4628,Z 74,A 147.1632,B 24.8785,C -2.5444,E1 24.857,E2 -63.0569} C_DIS
LIN {X -56.545,Y 31.0226,Z 74,A 144.6379,B 24.8777,C -2.5526,E1 24.8604,E2 -60.5377} C_DIS
LIN {X -55.3257,Y 33.1504,Z 74,A 141.9543,B 24.878,C -2.549,E1 24.8642,E2 -57.8317} C_DIS
LIN {X -52.4314,Y 37.5593,Z 74,A 137.2842,B 24.8768,C -2.5621,E1 24.8715,E2 -53.1697} C_DIS
LIN {X -49.7088,Y 41.095,Z 74,A 133.9394,B 24.8746,C -2.5844,E1 24.8773,E2 -49.8626} C_DIS
LIN {X -47.7101,Y 43.4,Z 74,A 130.744,B 24.8749,C -2.5817,E1 24.8832,E2 -46.6463} C_DIS
LIN {X -45.5958,Y 45.6169,Z 74,A 128.2356,B 24.8738,C -2.5924,E1 24.8881,E2 -44.1527} C_DIS
LIN {X -42.5988,Y 48.4266,Z 74,A 124.7092,B 24.8728,C -2.6032,E1 24.8953,E2 -40.6377} C_DIS
LIN {X -39.8469,Y 50.7148,Z 74,A 120.9289,B 24.8733,C -2.5981,E1 24.9036,E2 -36.831} C_DIS
LIN {X -37.6757,Y 52.3483,Z 74,A 118.2246,B 24.8733,C -2.5971,E1 24.9097,E2 -34.115} C_DIS
LIN {X -33.2176,Y 55.285,Z 74,A 114.136,B 24.8712,C -2.619,E1 24.9193,E2 -30.0656} C_DIS
LIN {X -30.6202,Y 56.7641,Z 74,A 111.6092,B 24.8705,C -2.6262,E1 24.9254,E2 -27.5486} C_DIS
LIN {X -28.5592,Y 57.8284,Z 74,A 109.2463,B 24.8708,C -2.6233,E1 24.9313,E2 -25.1725} C_DIS
LIN {X -24.6707,Y 59.5923,Z 74,A 105.549,B 24.8701,C -2.6307,E1 24.9408,E2 -21.4842} C_DIS
LIN {X -20.4958,Y 61.1529,Z 74,A 101.3164,B 24.8701,C -2.63,E1 24.9519,E2 -17.2415} C_DIS
LIN {X -16.4779,Y 62.3566,Z 74,A 98.087,B 24.8687,C -2.6444,E1 24.9605,E2 -14.0411} C_DIS
LIN {X -11.5054,Y 63.4616,Z 74,A 93.5789,B 24.8683,C -2.6486,E1 24.9728,E2 -9.5375} C_DIS
LIN {X -9.4078,Y 63.8071,Z 74,A 91.508,B 24.8685,C -2.646,E1 24.9785,E2 -7.4584} C_DIS
LIN {X -6.749,Y 64.1419,Z 74,A 89.1382,B 24.8684,C -2.6475,E1 24.9851,E2 -5.0909} C_DIS
LIN {X -2.1749,Y 64.4596,Z 74,A 85.4587,B 24.8674,C -2.6577,E1 24.9953,E2 -1.4344} C_DIS
LIN {X 1.6205,Y 64.4767,Z 74,A 81.6823,B 24.8682,C -2.6494,E1 25.0059,E2 2.3616} C_DIS
LIN {X 4.1146,Y 64.3651,Z 74,A 79.5019,B 24.8682,C -2.6503,E1 25.012,E2 4.5391} C_DIS
LIN {X 7.4773,Y 64.0611,Z 74,A 76.1934,B 24.8688,C -2.6431,E1 25.0212,E2 7.8626} C_DIS
LIN {X 10.6344,Y 63.6133,Z 74,A 73.6558,B 24.8683,C -2.6489,E1 25.0282,E2 10.384} C_DIS
LIN {X 13.2243,Y 63.1262,Z 74,A 71.2118,B 24.8686,C -2.6455,E1 25.0349,E2 12.8331} C_DIS
LIN {X 16.8288,Y 62.2618,Z 74,A 67.8989,B 24.8688,C -2.6432,E1 25.0438,E2 16.1466} C_DIS
LIN {X 19.0044,Y 61.6326,Z 74,A 65.7837,B 24.8692,C -2.6393,E1 25.0495,E2 18.2671} C_DIS
LIN {X 21.9691,Y 60.6392,Z 74,A 63.1709,B 24.8691,C -2.6407,E1 25.0564,E2 20.8714} C_DIS
LIN {X 24.9285,Y 59.4838,Z 74,A 60.6608,B 24.8686,C -2.6452,E1 25.0628,E2 23.3652} C_DIS
LIN {X 26.4851,Y 58.8071,Z 74,A 58.8578,B 24.8695,C -2.6366,E1 25.0675,E2 25.1841} C_DIS
LIN {X 30.5884,Y 56.7813,Z 74,A 54.7653,B 24.87,C -2.6309,E1 25.0777,E2 29.2791} C_DIS
LIN {X 32.3376,Y 55.8038,Z 74,A 53.0252,B 24.8702,C -2.6293,E1 25.0819,E2 31.0176} C_DIS
LIN {X 35.3781,Y 53.9273,Z 74,A 49.9347,B 24.8705,C -2.6265,E1 25.0892,E2 34.1049} C_DIS
LIN {X 38.3258,Y 51.8738,Z 74,A 46.7557,B 24.871,C -2.6215,E1 25.0964,E2 37.2847} C_DIS
LIN {X 40.0966,Y 50.5175,Z 74,A 44.1695,B 24.8727,C -2.6034,E1 25.1021,E2 39.9041} C_DIS
LIN {X 43.7286,Y 47.4086,Z 74,A 40.4144,B 24.8724,C -2.607,E1 25.1099,E2 43.6358} C_DIS
LIN {X 46.119,Y 45.0867,Z 74,A 37.3096,B 24.8733,C -2.5973,E1 25.1161,E2 46.7504} C_DIS
LIN {X 49.1482,Y 41.7636,Z 74,A 33.5791,B 24.8736,C -2.5948,E1 25.123,E2 50.47} C_DIS
LIN {X 51.1073,Y 39.3418,Z 74,A 30.821,B 24.8742,C -2.5886,E1 25.1278,E2 53.2301} C_DIS
LIN {X 52.6785,Y 37.213,Z 74,A 28.4789,B 24.8747,C -2.583,E1 25.1316,E2 55.574} C_DIS
LIN {X 54.1984,Y 34.9612,Z 74,A 26.002,B 24.8755,C -2.5753,E1 25.1354,E2 58.0567} C_DIS
LIN {X 55.5328,Y 32.8,Z 74,A 23.5405,B 24.8765,C -2.5643,E1 25.139,E2 60.5315} C_DIS
LIN {X 57.7272,Y 28.7632,Z 74,A 20.0645,B 24.8761,C -2.5685,E1 25.1435,E2 63.9794} C_DIS
LIN {X 59.2596,Y 25.4588,Z 74,A 16.0898,B 24.8788,C -2.5408,E1 25.1481,E2 67.9978} C_DIS
LIN {X 60.5955,Y 22.0889,Z 74,A 13.4257,B 24.8784,C -2.5456,E1 25.1507,E2 70.636} C_DIS
LIN {X 61.6651,Y 18.8997,Z 74,A 9.8311,B 24.8807,C -2.5214,E1 25.1538,E2 74.2673} C_DIS
LIN {X 62.5705,Y 15.6463,Z 74,A 7.3245,B 24.8803,C -2.5249,E1 25.1555,E2 76.7513} C_DIS
LIN {X 63.2415,Y 12.6629,Z 74,A 4.0762,B 24.8824,C -2.5031,E1 25.1574,E2 80.0321} C_DIS
LIN {X 64.1327,Y 6.8373,Z 74,A -0.0248,B 24.8812,C -2.5158,E1 25.1589,E2 84.079} C_DIS
LIN {X 64.3123,Y 4.8719,Z 74,A -2.2266,B 24.8828,C -2.4988,E1 25.1594,E2 86.3079} C_DIS
LIN {X 64.4939,Y -0.5327,Z 74,A -6.5699,B 24.8831,C -2.4954,E1 25.1598,E2 90.6332} C_DIS
LIN {X 64.38,Y -3.8806,Z 74,A -10.4426,B 24.8861,C -2.463,E1 25.1593,E2 94.5595} C_DIS
LIN {X 64.128,Y -6.8821,Z 74,A -13.0306,B 24.8867,C -2.4567,E1 25.1585,E2 97.147} C_DIS
LIN {X 63.5268,Y -11.1425,Z 74,A -16.7172,B 24.8875,C -2.4481,E1 25.1569,E2 100.8323} C_DIS
LIN {X 62.9527,Y -14.0276,Z 74,A -19.0305,B 24.8875,C -2.4476,E1 25.1556,E2 103.1335} C_DIS
LIN {X 61.5479,Y -19.2776,Z 74,A -23.5605,B 24.8882,C -2.4402,E1 25.1522,E2 107.6548} C_DIS
LIN {X 60.2936,Y -22.9001,Z 74,A -26.9714,B 24.8892,C -2.4296,E1 25.149,E2 111.0716} C_DIS
LIN {X 59.5813,Y -24.6971,Z 74,A -29.3076,B 24.8911,C -2.4087,E1 25.1465,E2 113.4445} C_DIS
LIN {X 57.4339,Y -29.3442,Z 74,A -33.3854,B 24.8913,C -2.4072,E1 25.1416,E2 117.5038} C_DIS
LIN {X 55.0835,Y -33.5492,Z 74,A -37.4982,B 24.892,C -2.3992,E1 25.1359,E2 121.6142} C_DIS
LIN {X 53.67,Y -35.7683,Z 74,A -40.3465,B 24.8937,C -2.3798,E1 25.1315,E2 124.4941} C_DIS
LIN {X 51.6042,Y -38.6879,Z 74,A -43.487,B 24.8944,C -2.3722,E1 25.1263,E2 127.6374} C_DIS
LIN {X 48.4429,Y -42.5801,Z 74,A -47.0389,B 24.8934,C -2.3834,E1 25.1201,E2 131.1466} C_DIS
LIN {X 45.7852,Y -45.4254,Z 74,A -51.0988,B 24.8955,C -2.3598,E1 25.1122,E2 135.2445} C_DIS
LIN {X 44.0584,Y -47.1016,Z 74,A -54.2369,B 24.8981,C -2.3302,E1 25.1057,E2 138.4399} C_DIS
LIN {X 40.9835,Y -49.8014,Z 74,A -56.4942,B 24.8958,C -2.356,E1 25.101,E2 140.6274} C_DIS
LIN {X 38.2495,Y -51.9302,Z 74,A -60.1698,B 24.8977,C -2.3349,E1 25.0927,E2 144.3398} C_DIS
LIN {X 35.2227,Y -54.0287,Z 74,A -63.1632,B 24.8977,C -2.3353,E1 25.0858,E2 147.3221} C_DIS
LIN {X 33.1416,Y -55.3309,Z 74,A -65.2856,B 24.8979,C -2.3327,E1 25.0808,E2 149.4441} C_DIS
LIN {X 29.542,Y -57.3329,Z 74,A -69.4163,B 24.8994,C -2.3151,E1 25.0705,E2 153.6046} C_DIS
LIN {X 24.437,Y -59.6874,Z 74,A -74.3802,B 24.9,C -2.3085,E1 25.0578,E2 158.5722} C_DIS
LIN {X 20.5572,Y -61.1322,Z 74,A -77.8602,B 24.9,C -2.3085,E1 25.0487,E2 162.0451} C_DIS
LIN {X 17.3755,Y -62.1118,Z 74,A -80.678,B 24.9,C -2.3085,E1 25.0411,E2 164.858} C_DIS
LIN {X 14.3517,Y -62.8792,Z 74,A -83.3074,B 24.9,C -2.3092,E1 25.034,E2 167.4821} C_DIS
LIN {X 10.2441,Y -63.6775,Z 74,A -87.1476,B 24.9005,C -2.3034,E1 25.0234,E2 171.3318} C_DIS
LIN {X 6.2512,Y -64.1932,Z 74,A -90.5447,B 24.9003,C -2.3054,E1 25.014,E2 174.7217} C_DIS
LIN {X 3.344,Y -64.4096,Z 74,A -94.2321,B 24.9025,C -2.2795,E1 25.0036,E2 178.4693} C_DIS
LIN {X 3.344,Y -64.4096,Z 74,A -94.2321,B 24.9025,C -2.2795,E1 25.0036,E2 178.4693} C_DIS
Enddeposition()
LIN {X 0.3989,Y -63.5613,Z 74,A -94.5373,B 24.8966,C -2.3474,E1 25.0032,E2 178.6132} C_DIS
Startdeposition()
$VEL.CP = VEL_PRINT
LIN {X 4.0543,Y -63.4437,Z 74,A -91.219,B 24.8965,C -2.3489,E1 25.0124,E2 175.2923} C_DIS
LIN {X 7.0518,Y -63.1813,Z 74,A -88.6332,B 24.8966,C -2.3475,E1 25.0196,E2 172.7116} C_DIS
LIN {X 10.8349,Y -62.643,Z 74,A -84.9284,B 24.8958,C -2.356,E1 25.0299,E2 168.99} C_DIS
LIN {X 14.0365,Y -62.0044,Z 74,A -82.1128,B 24.8958,C -2.3556,E1 25.0376,E2 166.179} C_DIS
LIN {X 16.5646,Y -61.3767,Z 74,A -80.0292,B 24.8962,C -2.3518,E1 25.0432,E2 164.1077} C_DIS
LIN {X 19.9293,Y -60.3681,Z 74,A -76.6822,B 24.8955,C -2.3597,E1 25.0521,E2 160.7479} C_DIS
LIN {X 23.6563,Y -59.0067,Z 74,A -72.7348,B 24.8943,C -2.3735,E1 25.0625,E2 156.7765} C_DIS
LIN {X 27.2872,Y -57.4192,Z 74,A -69.8879,B 24.8954,C -2.3613,E1 25.0696,E2 153.9655} C_DIS
LIN {X 31.2027,Y -55.3889,Z 74,A -65.6312,B 24.8942,C -2.3748,E1 25.0802,E2 149.6888} C_DIS
LIN {X 33.4804,Y -54.0426,Z 74,A -63.5846,B 24.8945,C -2.3709,E1 25.085,E2 147.6578} C_DIS
LIN {X 35.759,Y -52.5623,Z 74,A -60.7044,B 24.8931,C -2.3863,E1 25.0918,E2 144.7508} C_DIS
LIN {X 38.4433,Y -50.6318,Z 74,A -57.6991,B 24.8925,C -2.393,E1 25.0986,E2 141.7403} C_DIS
LIN {X 40.9347,Y -48.6414,Z 74,A -55.0583,B 24.8925,C -2.3935,E1 25.1042,E2 139.1084} C_DIS
LIN {X 43.1411,Y -46.6932,Z 74,A -52.3331,B 24.8918,C -2.4014,E1 25.1099,E2 136.3754} C_DIS
LIN {X 45.3054,Y -44.5973,Z 74,A -49.3259,B 24.8905,C -2.4152,E1 25.1159,E2 133.3482} C_DIS
LIN {X 47.6779,Y -42.0524,Z 74,A -46.4862,B 24.8905,C -2.4156,E1 25.1212,E2 130.5203} C_DIS
LIN {X 50.9291,Y -38.0492,Z 74,A -41.5147,B 24.8886,C -2.436,E1 25.1298,E2 125.5239} C_DIS
LIN {X 52.9576,Y -35.1714,Z 74,A -38.7712,B 24.8888,C -2.4337,E1 25.1341,E2 122.7993} C_DIS
LIN {X 54.6272,Y -32.5176,Z 74,A -35.0429,B 24.886,C -2.4648,E1 25.1396,E2 119.0164} C_DIS
LIN {X 56.3149,Y -29.4981,Z 74,A -32.9159,B 24.8875,C -2.4484,E1 25.1423,E2 116.9394} C_DIS
LIN {X 57.3027,Y -27.5296,Z 74,A -30.6623,B 24.8863,C -2.4611,E1 25.1451,E2 114.6679} C_DIS
LIN {X 58.8469,Y -24.0529,Z 74,A -27.607,B 24.8863,C -2.4618,E1 25.1485,E2 111.6276} C_DIS
LIN {X 59.8033,Y -21.5662,Z 74,A -24.7017,B 24.8844,C -2.4821,E1 25.1513,E2 108.6907} C_DIS
LIN {X 61.007,Y -17.8795,Z 74,A -21.0256,B 24.8829,C -2.4976,E1 25.1543,E2 104.999} C_DIS
LIN {X 62.0464,Y -13.8503,Z 74,A -17.8315,B 24.8832,C -2.4949,E1 25.1564,E2 101.8296} C_DIS
LIN {X 62.6262,Y -10.9337,Z 74,A -14.5752,B 24.881,C -2.5183,E1 25.158,E2 98.5372} C_DIS
LIN {X 63.2065,Y -6.8163,Z 74,A -11.4732,B 24.8814,C -2.5134,E1 25.159,E2 95.465} C_DIS
LIN {X 63.5557,Y -1.51,Z 74,A -6.6682,B 24.88,C -2.5289,E1 25.1598,E2 90.652} C_DIS
LIN {X 63.5186,Y 2.6245,Z 74,A -3.1238,B 24.8793,C -2.536,E1 25.1596,E2 87.1119} C_DIS
LIN {X 63.3576,Y 5.228,Z 74,A -0.7094,B 24.8784,C -2.545,E1 25.1591,E2 84.6905} C_DIS
LIN {X 63.0933,Y 7.8014,Z 74,A 1.9168,B 24.877,C -2.5598,E1 25.1582,E2 82.0448} C_DIS
LIN {X 62.5106,Y 11.5766,Z 74,A 5.0727,B 24.8767,C -2.5631,E1 25.1568,E2 78.8997} C_DIS
LIN {X 61.936,Y 14.3326,Z 74,A 7.5674,B 24.876,C -2.5697,E1 25.1553,E2 76.4037} C_DIS
LIN {X 61.2544,Y 17.0147,Z 74,A 10.274,B 24.8748,C -2.5826,E1 25.1533,E2 73.6823} C_DIS
LIN {X 60.3048,Y 20.121,Z 74,A 13.0513,B 24.8743,C -2.5874,E1 25.1509,E2 70.9093} C_DIS
LIN {X 59.2994,Y 22.917,Z 74,A 16.5879,B 24.8714,C -2.6171,E1 25.1473,E2 67.3223} C_DIS
LIN {X 57.8811,Y 26.2926,Z 74,A 18.9308,B 24.8729,C -2.602,E1 25.1447,E2 65.0279} C_DIS
LIN {X 56.5992,Y 28.9485,Z 74,A 21.3588,B 24.8727,C -2.6035,E1 25.1417,E2 62.6093} C_DIS
LIN {X 54.5432,Y 32.6598,Z 74,A 25.526,B 24.8709,C -2.6222,E1 25.136,E2 58.4195} C_DIS
LIN {X 52.9015,Y 35.2565,Z 74,A 28.1957,B 24.8705,C -2.6267,E1 25.1319,E2 55.7524} C_DIS
LIN {X 51.1656,Y 37.7309,Z 74,A 31.2467,B 24.869,C -2.6415,E1 25.1268,E2 52.681} C_DIS
LIN {X 48.9837,Y 40.5228,Z 74,A 34.1495,B 24.869,C -2.6417,E1 25.1218,E2 49.7913} C_DIS
LIN {X 46.8227,Y 43.0014,Z 74,A 36.8288,B 24.869,C -2.6413,E1 25.1168,E2 47.1249} C_DIS
LIN {X 45.0426,Y 44.8634,Z 74,A 39.199,B 24.8684,C -2.6474,E1 25.1122,E2 44.7504} C_DIS
LIN {X 43.4902,Y 46.3691,Z 74,A 41.179,B 24.8679,C -2.6521,E1 25.1082,E2 42.7674} C_DIS
LIN {X 41.5677,Y 48.1012,Z 74,A 43.6232,B 24.8672,C -2.6594,E1 25.103,E2 40.3157} C_DIS
LIN {X 38.6242,Y 50.4947,Z 74,A 47.0738,B 24.8665,C -2.6663,E1 25.0955,E2 36.8616} C_DIS
LIN {X 35.9002,Y 52.4667,Z 74,A 49.7876,B 24.8668,C -2.6637,E1 25.0893,E2 34.1633} C_DIS
LIN {X 34.1705,Y 53.6088,Z 74,A 51.9749,B 24.8657,C -2.6742,E1 25.0841,E2 31.9581} C_DIS
LIN {X 31.4732,Y 55.2356,Z 74,A 54.6933,B 24.8656,C -2.6754,E1 25.0776,E2 29.2453} C_DIS
LIN {X 28.1302,Y 57.0104,Z 74,A 58.0191,B 24.8654,C -2.6777,E1 25.0693,E2 25.9231} C_DIS
LIN {X 25.767,Y 58.1179,Z 74,A 60.4682,B 24.8649,C -2.6826,E1 25.0631,E2 23.4686} C_DIS
LIN {X 23.0318,Y 59.2539,Z 74,A 63.0158,B 24.8649,C -2.6825,E1 25.0565,E2 20.927} C_DIS
LIN {X 18.5703,Y 60.8005,Z 74,A 67.1749,B 24.8648,C -2.6837,E1 25.0455,E2 16.7732} C_DIS
LIN {X 16.4637,Y 61.404,Z 74,A 69.4166,B 24.864,C -2.6911,E1 25.0394,E2 14.5174} C_DIS
LIN {X 13.0652,Y 62.2163,Z 74,A 72.4997,B 24.864,C -2.6911,E1 25.031,E2 11.4384} C_DIS
LIN {X 9.9253,Y 62.7935,Z 74,A 75.3421,B 24.864,C -2.6913,E1 25.0232,E2 8.5985} C_DIS
LIN {X 5.5724,Y 63.3286,Z 74,A 79.3006,B 24.864,C -2.6921,E1 25.0123,E2 4.6411} C_DIS
LIN {X 2.4239,Y 63.5272,Z 74,A 82.1474,B 24.864,C -2.6921,E1 25.0043,E2 1.7953} C_DIS
LIN {X -0.171,Y 63.5728,Z 74,A 84.6599,B 24.8636,C -2.6954,E1 24.9973,E2 -0.7251} C_DIS
LIN {X -4.6047,Y 63.4065,Z 74,A 88.4507,B 24.8642,C -2.6894,E1 24.9867,E2 -4.5028} C_DIS
LIN {X -7.4874,Y 63.1303,Z 74,A 91.0318,B 24.8644,C -2.6874,E1 24.9796,E2 -7.0806} C_DIS
LIN {X -10.2667,Y 62.7386,Z 74,A 93.5084,B 24.8647,C -2.6846,E1 24.9728,E2 -9.5526} C_DIS
LIN {X -11.9673,Y 62.4362,Z 74,A 96.0044,B 24.8627,C -2.7036,E1 24.9658,E2 -12.0967} C_DIS
LIN {X -15.3804,Y 61.6849,Z 74,A 98.1927,B 24.8651,C -2.6801,E1 24.96,E2 -14.2319} C_DIS
LIN {X -17.7568,Y 61.0434,Z 74,A 101.3939,B 24.8632,C -2.6986,E1 24.9513,E2 -17.4825} C_DIS
LIN {X -21.0448,Y 59.9884,Z 74,A 103.5809,B 24.8656,C -2.6753,E1 24.9456,E2 -19.6181} C_DIS
LIN {X -23.6662,Y 59.0043,Z 74,A 106.1594,B 24.8658,C -2.6731,E1 24.9389,E2 -22.1968} C_DIS
LIN {X -26.2234,Y 57.9123,Z 74,A 108.2893,B 24.867,C -2.6617,E1 24.9335,E2 -24.3046} C_DIS
LIN {X -27.9216,Y 57.1139,Z 74,A 110.5024,B 24.8661,C -2.6698,E1 24.9279,E2 -26.5428} C_DIS
LIN {X -30.8583,Y 55.5813,Z 74,A 113.2003,B 24.8672,C -2.659,E1 24.9213,E2 -29.2224} C_DIS
LIN {X -32.5916,Y 54.5835,Z 74,A 115.364,B 24.8668,C -2.6631,E1 24.9161,E2 -31.4026} C_DIS
LIN {X -35.87,Y 52.4872,Z 74,A 118.6938,B 24.8679,C -2.6529,E1 24.9083,E2 -34.7188} C_DIS
LIN {X -38.1686,Y 50.8394,Z 74,A 122.2819,B 24.8663,C -2.6688,E1 24.9002,E2 -38.3577} C_DIS
LIN {X -41.1351,Y 48.4707,Z 74,A 124.695,B 24.869,C -2.6409,E1 24.8951,E2 -40.7136} C_DIS
LIN {X -44.9986,Y 44.9079,Z 74,A 129.9878,B 24.869,C -2.641,E1 24.8844,E2 -46.0284} C_DIS
LIN {X -48.547,Y 41.0455,Z 74,A 134.0397,B 24.8715,C -2.6159,E1 24.8769,E2 -50.0384} C_DIS
LIN {X -51.0289,Y 37.9163,Z 74,A 137.8838,B 24.872,C -2.6112,E1 24.8704,E2 -53.8896} C_DIS
LIN {X -52.3703,Y 36.0406,Z 74,A 139.7619,B 24.8729,C -2.6017,E1 24.8674,E2 -55.7542} C_DIS
LIN {X -54.6342,Y 32.5057,Z 74,A 143.7734,B 24.8735,C -2.5956,E1 24.8614,E2 -59.7716} C_DIS
LIN {X -56.9404,Y 28.2715,Z 74,A 147.8005,B 24.8753,C -2.5769,E1 24.8562,E2 -63.7753} C_DIS
LIN {X -58.7398,Y 24.3158,Z 74,A 152.0206,B 24.8759,C -2.5711,E1 24.8514,E2 -68.0047} C_DIS
LIN {X -59.7473,Y 21.7198,Z 74,A 154.6148,B 24.8765,C -2.5651,E1 24.8488,E2 -70.5992} C_DIS
LIN {X -60.4387,Y 19.7148,Z 74,A 157.2047,B 24.8758,C -2.5723,E1 24.8466,E2 -73.2212} C_DIS
LIN {X -61.6416,Y 15.5526,Z 74,A 161.0518,B 24.8771,C -2.559,E1 24.8438,E2 -77.059} C_DIS
LIN {X -62.437,Y 11.9631,Z 74,A 163.7031,B 24.8793,C -2.5359,E1 24.8424,E2 -79.6707} C_DIS
LIN {X -62.904,Y 9.2,Z 74,A 166.4088,B 24.8797,C -2.5314,E1 24.8412,E2 -82.3816} C_DIS
LIN {X -63.2856,Y 6.0384,Z 74,A 169.2405,B 24.8806,C -2.5216,E1 24.8403,E2 -85.2069} C_DIS
LIN {X -63.5125,Y 2.7656,Z 74,A 172.2255,B 24.8815,C -2.5128,E1 24.8399,E2 -88.1887} C_DIS
LIN {X -63.5724,Y 0.0854,Z 74,A 174.6607,B 24.8822,C -2.5055,E1 24.8398,E2 -90.6212} C_DIS
LIN {X -63.5143,Y -2.7233,Z 74,A 177.0144,B 24.8832,C -2.4941,E1 24.84,E2 -92.9618} C_DIS
LIN {X -63.3276,Y -5.5828,Z 74,A 179.3915,B 24.8844,C -2.4821,E1 24.8405,E2 -95.3245} C_DIS
LIN {X -63.1527,Y -7.2958,Z 74,A -178.7851,B 24.8844,C -2.4824,E1 24.841,E2 -97.1596} C_DIS
LIN {X -62.757,Y -10.1563,Z 74,A -175.9045,B 24.8846,C -2.4797,E1 24.8422,E2 -100.0509} C_DIS
LIN {X -62.2353,Y -12.9727,Z 74,A -173.3391,B 24.8854,C -2.4715,E1 24.8436,E2 -102.6119} C_DIS
LIN {X -61.7625,Y -15.0624,Z 74,A -171.1622,B 24.8854,C -2.4704,E1 24.8451,E2 -104.799} C_DIS
LIN {X -60.2268,Y -20.3506,Z 74,A -166.4705,B 24.8873,C -2.4505,E1 24.8489,E2 -109.4699} C_DIS
LIN {X -58.6726,Y -24.4758,Z 74,A -162.4661,B 24.8883,C -2.4397,E1 24.8529,E2 -113.471} C_DIS
LIN {X -57.457,Y -27.2086,Z 74,A -159.7633,B 24.889,C -2.4323,E1 24.8561,E2 -116.1709} C_DIS
LIN {X -56.6007,Y -28.9457,Z 74,A -157.9293,B 24.8892,C -2.4293,E1 24.8584,E2 -118.0077} C_DIS
LIN {X -55.1044,Y -31.7016,Z 74,A -155.2583,B 24.8902,C -2.4187,E1 24.862,E2 -120.6675} C_DIS
LIN {X -53.9201,Y -33.6765,Z 74,A -152.4311,B 24.8893,C -2.4284,E1 24.8663,E2 -123.5321} C_DIS
LIN {X -51.4932,Y -37.2834,Z 74,A -149.0574,B 24.8912,C -2.4078,E1 24.8716,E2 -126.8732} C_DIS
LIN {X -49.5999,Y -39.7674,Z 74,A -146.1303,B 24.8916,C -2.4034,E1 24.8767,E2 -129.8037} C_DIS
LIN {X -47.3089,Y -42.466,Z 74,A -143.116,B 24.8926,C -2.3927,E1 24.8822,E2 -132.8061} C_DIS
LIN {X -44.8618,Y -45.0439,Z 74,A -139.692,B 24.8928,C -2.3905,E1 24.8889,E2 -136.2393} C_DIS
LIN {X -41.3864,Y -48.2566,Z 74,A -135.6158,B 24.8939,C -2.3782,E1 24.8973,E2 -140.3027} C_DIS
LIN {X -39.2845,Y -49.9824,Z 74,A -133.2265,B 24.8944,C -2.3725,E1 24.9025,E2 -142.6874} C_DIS
LIN {X -36.4497,Y -52.0856,Z 74,A -130.0758,B 24.8949,C -2.3666,E1 24.9096,E2 -145.8349} C_DIS
LIN {X -34.0291,Y -53.6995,Z 74,A -127.4728,B 24.8953,C -2.3621,E1 24.9157,E2 -148.4357} C_DIS
LIN {X -31.2759,Y -55.3481,Z 74,A -124.4291,B 24.8953,C -2.3612,E1 24.923,E2 -151.4865} C_DIS
LIN {X -28.8839,Y -56.6323,Z 74,A -122.0194,B 24.8957,C -2.3574,E1 24.929,E2 -153.8937} C_DIS
LIN {X -26.9151,Y -57.594,Z 74,A -119.9792,B 24.8958,C -2.3565,E1 24.9341,E2 -155.9369} C_DIS
LIN {X -24.7122,Y -58.573,Z 74,A -116.9397,B 24.8943,C -2.3731,E1 24.9421,E2 -159.0228} C_DIS
LIN {X -21.4605,Y -59.8419,Z 74,A -114.7316,B 24.8964,C -2.3498,E1 24.9477,E2 -161.1801} C_DIS
LIN {X -17.8866,Y -61.0049,Z 74,A -111.2702,B 24.8964,C -2.3489,E1 24.957,E2 -164.6455} C_DIS
LIN {X -15.0418,Y -61.7676,Z 74,A -108.7963,B 24.897,C -2.3435,E1 24.9636,E2 -167.11} C_DIS
LIN {X -12.4652,Y -62.3395,Z 74,A -106.3771,B 24.897,C -2.3433,E1 24.9702,E2 -169.5318} C_DIS
LIN {X -10.063,Y -62.7718,Z 74,A -103.9233,B 24.8965,C -2.3483,E1 24.977,E2 -171.9999} C_DIS
LIN {X -7.0617,Y -63.1801,Z 74,A -101.2475,B 24.8967,C -2.3467,E1 24.9845,E2 -174.6736} C_DIS
LIN {X -4.0549,Y -63.4437,Z 74,A -98.8255,B 24.8973,C -2.3399,E1 24.9912,E2 -177.0805} C_DIS
LIN {X -1.0732,Y -63.5637,Z 74,A -96.1394,B 24.8973,C -2.3402,E1 24.9987,E2 -179.7677} C_DIS
LIN {X 0.3989,Y -63.5613,Z 74,A -94.5363,B 24.8966,C -2.3469,E1 25.0032,E2 -181.3868} C_DIS
Enddeposition()
LIN {X 0.3989,Y -63.5613,Z 74,A -94.5363,B 24.8966,C -2.3469,E1 25.0032,E2 -181.3868} C_DIS
Startdeposition()
$VEL.CP = VEL_PRINT
LIN {X -0.9422,Y -62.6426,Z 74,A -97.1386,B 24.898,C -2.3317,E1 24.9958,E2 -178.7484} C_DIS
LIN {X -3.8055,Y -62.5346,Z 74,A -99.6279,B 24.8978,C -2.3344,E1 24.9889,E2 -176.2648} C_DIS
LIN {X -6.3371,Y -62.3283,Z 74,A -101.8951,B 24.8976,C -2.3358,E1 24.9826,E2 -173.9996} C_DIS
LIN {X -8.7767,Y -62.0316,Z 74,A -104.2963,B 24.8979,C -2.3329,E1 24.9759,E2 -171.5898} C_DIS
LIN {X -11.5622,Y -61.5739,Z 74,A -106.7553,B 24.8976,C -2.3363,E1 24.9692,E2 -169.1366} C_DIS
LIN {X -14.0591,Y -61.0515,Z 74,A -109.0647,B 24.8974,C -2.3379,E1 24.9629,E2 -166.828} C_DIS
LIN {X -16.5215,Y -60.4319,Z 74,A -111.5631,B 24.8977,C -2.3355,E1 24.9561,E2 -164.3202} C_DIS
LIN {X -19.5578,Y -59.519,Z 74,A -114.3423,B 24.8972,C -2.3401,E1 24.9487,E2 -161.5471} C_DIS
LIN {X -23.2982,Y -58.1572,Z 74,A -118.0092,B 24.897,C -2.3429,E1 24.9391,E2 -157.8791} C_DIS
LIN {X -26.1429,Y -56.935,Z 74,A -120.8229,B 24.8967,C -2.3463,E1 24.9319,E2 -155.0668} C_DIS
LIN {X -28.828,Y -55.6239,Z 74,A -123.5825,B 24.8965,C -2.349,E1 24.925,E2 -152.3065} C_DIS
LIN {X -30.9604,Y -54.4654,Z 74,A -125.758,B 24.8961,C -2.3529,E1 24.9197,E2 -150.1339} C_DIS
LIN {X -33.2071,Y -53.1247,Z 74,A -128.2128,B 24.8959,C -2.3551,E1 24.9139,E2 -147.6768} C_DIS
LIN {X -35.3635,Y -51.7149,Z 74,A -130.921,B 24.8962,C -2.3518,E1 24.9076,E2 -144.9517} C_DIS
LIN {X -38.0734,Y -49.7534,Z 74,A -133.6578,B 24.8952,C -2.3635,E1 24.9015,E2 -142.2329} C_DIS
LIN {X -40.3627,Y -47.9157,Z 74,A -136.3348,B 24.8947,C -2.3685,E1 24.8957,E2 -139.5578} C_DIS
LIN {X -42.3441,Y -46.1727,Z 74,A -139.3779,B 24.8954,C -2.361,E1 24.8894,E2 -136.4844} C_DIS
LIN {X -45.3811,Y -43.1931,Z 74,A -142.5405,B 24.8934,C -2.3832,E1 24.8832,E2 -133.3615} C_DIS
LIN {X -47.2268,Y -41.1652,Z 74,A -145.2358,B 24.8932,C -2.3852,E1 24.8782,E2 -130.6587} C_DIS
LIN {X -49.1366,Y -38.8656,Z 74,A -147.9103,B 24.8926,C -2.3926,E1 24.8735,E2 -127.9896} C_DIS
LIN {X -50.5959,Y -36.9459,Z 74,A -150.2354,B 24.8923,C -2.3956,E1 24.8696,E2 -125.6604} C_DIS
LIN {X -52.0802,Y -34.8243,Z 74,A -152.3901,B 24.8914,C -2.4056,E1 24.8662,E2 -123.5188} C_DIS
LIN {X -53.4226,Y -32.7264,Z 74,A -154.7748,B 24.8911,C -2.4094,E1 24.8627,E2 -121.1311} C_DIS
LIN {X -54.7072,Y -30.5298,Z 74,A -157.1851,B 24.8906,C -2.4139,E1 24.8594,E2 -118.7191} C_DIS
LIN {X -55.9367,Y -28.2159,Z 74,A -159.5636,B 24.89,C -2.4207,E1 24.8563,E2 -116.3441} C_DIS
LIN {X -57.0017,Y -25.9967,Z 74,A -161.821,B 24.8895,C -2.4269,E1 24.8536,E2 -114.089} C_DIS
LIN {X -57.9932,Y -23.7011,Z 74,A -164.3747,B 24.8893,C -2.4284,E1 24.8509,E2 -111.5248} C_DIS
LIN {X -59.1704,Y -20.5871,Z 74,A -167.2269,B 24.8882,C -2.4408,E1 24.8482,E2 -108.686} C_DIS
LIN {X -59.989,Y -18.0646,Z 74,A -169.8712,B 24.8879,C -2.4439,E1 24.846,E2 -106.034} C_DIS
LIN {X -60.8667,Y -14.8389,Z 74,A -172.7328,B 24.8867,C -2.4567,E1 24.844,E2 -103.1863} C_DIS
LIN {X -61.455,Y -12.1796,Z 74,A -175.2591,B 24.8861,C -2.4636,E1 24.8425,E2 -100.6616} C_DIS
LIN {X -61.9153,Y -9.5622,Z 74,A -177.6668,B 24.8853,C -2.4715,E1 24.8414,E2 -98.2586} C_DIS
LIN {X -62.2518,Y -7.0505,Z 74,A 179.9608,B 24.8848,C -2.4777,E1 24.8406,E2 -95.8867} C_DIS
LIN {X -62.4893,Y -4.4822,Z 74,A 177.6075,B 24.8841,C -2.4852,E1 24.8401,E2 -93.5372} C_DIS
LIN {X -62.6225,Y -1.8375,Z 74,A 175.1703,B 24.8834,C -2.4925,E1 24.8398,E2 -91.1029} C_DIS
LIN {X -62.6416,Y 0.9993,Z 74,A 172.6062,B 24.8826,C -2.5013,E1 24.8398,E2 -88.5443} C_DIS
LIN {X -62.5807,Y 2.9427,Z 74,A 170.6924,B 24.8823,C -2.5044,E1 24.8401,E2 -86.6265} C_DIS
LIN {X -62.3883,Y 5.7138,Z 74,A 168.2752,B 24.8813,C -2.5147,E1 24.8406,E2 -84.2194} C_DIS
LIN {X -62.1064,Y 8.2327,Z 74,A 165.8799,B 24.8807,C -2.5206,E1 24.8414,E2 -81.8239} C_DIS
LIN {X -61.72,Y 10.7562,Z 74,A 163.5151,B 24.8801,C -2.5274,E1 24.8425,E2 -79.4612} C_DIS
LIN {X -61.0679,Y 13.9874,Z 74,A 160.4742,B 24.8792,C -2.5364,E1 24.8442,E2 -76.4239} C_DIS
LIN {X -60.583,Y 15.9621,Z 74,A 158.326,B 24.8792,C -2.5369,E1 24.8457,E2 -74.2643} C_DIS
LIN {X -59.7001,Y 18.9982,Z 74,A 155.5452,B 24.8781,C -2.5478,E1 24.848,E2 -71.4937} C_DIS
LIN {X -58.7878,Y 21.6559,Z 74,A 152.9671,B 24.8774,C -2.5555,E1 24.8504,E2 -68.9192} C_DIS
LIN {X -57.738,Y 24.3161,Z 74,A 150.2645,B 24.8768,C -2.5618,E1 24.8533,E2 -66.2166} C_DIS
LIN {X -56.5368,Y 26.9918,Z 74,A 147.8961,B 24.8755,C -2.5755,E1 24.856,E2 -63.868} C_DIS
LIN {X -54.8095,Y 30.3451,Z 74,A 144.3716,B 24.8746,C -2.584,E1 24.8606,E2 -60.3453} C_DIS
LIN {X -53.3575,Y 32.8323,Z 74,A 141.3163,B 24.8746,C -2.5836,E1 24.865,E2 -57.2732} C_DIS
LIN {X -51.4026,Y 35.815,Z 74,A 138.5375,B 24.8729,C -2.6015,E1 24.8693,E2 -54.5233} C_DIS
LIN {X -49.8867,Y 37.8996,Z 74,A 135.7,B 24.8732,C -2.5988,E1 24.8741,E2 -51.6656} C_DIS
LIN {X -47.6887,Y 40.6292,Z 74,A 132.1482,B 24.873,C -2.6005,E1 24.8805,E2 -48.1015} C_DIS
LIN {X -44.8313,Y 43.7634,Z 74,A 128.7788,B 24.8712,C -2.6195,E1 24.8869,E2 -44.7628} C_DIS
LIN {X -43.2085,Y 45.3663,Z 74,A 126.378,B 24.8712,C -2.6184,E1 24.8917,E2 -42.3494} C_DIS
LIN {X -40.4986,Y 47.8,Z 74,A 123.0163,B 24.8706,C -2.6252,E1 24.8988,E2 -38.9908} C_DIS
LIN {X -37.6244,Y 50.0934,Z 74,A 120.1245,B 24.869,C -2.6413,E1 24.9051,E2 -36.1269} C_DIS
LIN {X -35.4484,Y 51.6575,Z 74,A 117.5308,B 24.8688,C -2.6433,E1 24.9111,E2 -33.5292} C_DIS
LIN {X -33.6865,Y 52.8223,Z 74,A 115.336,B 24.8689,C -2.6419,E1 24.9163,E2 -31.3237} C_DIS
LIN {X -31.099,Y 54.3858,Z 74,A 112.2422,B 24.8691,C -2.6403,E1 24.9238,E2 -28.217} C_DIS
LIN {X -27.4673,Y 56.3083,Z 74,A 109.023,B 24.8674,C -2.6569,E1 24.9317,E2 -25.0288} C_DIS
LIN {X -24.6707,Y 57.5885,Z 74,A 106.1519,B 24.8672,C -2.6598,E1 24.939,E2 -22.1578} C_DIS
LIN {X -21.6985,Y 58.7722,Z 74,A 103.2231,B 24.8668,C -2.6636,E1 24.9466,E2 -19.2317} C_DIS
LIN {X -18.7842,Y 59.7675,Z 74,A 100.3177,B 24.8666,C -2.6651,E1 24.9544,E2 -16.3247} C_DIS
LIN {X -15.822,Y 60.619,Z 74,A 97.9839,B 24.8653,C -2.6779,E1 24.9606,E2 -14.0176} C_DIS
LIN {X -13.0142,Y 61.2837,Z 74,A 95.007,B 24.8658,C -2.6733,E1 24.9687,E2 -11.0259} C_DIS
LIN {X -10.5463,Y 61.7557,Z 74,A 92.7916,B 24.8655,C -2.6767,E1 24.9748,E2 -8.8164} C_DIS
LIN {X -8.1225,Y 62.1206,Z 74,A 90.5835,B 24.8652,C -2.6789,E1 24.9809,E2 -6.6116} C_DIS
LIN {X -5.6319,Y 62.3958,Z 74,A 88.161,B 24.8654,C -2.6773,E1 24.9876,E2 -4.184} C_DIS
LIN {X -2.7103,Y 62.5907,Z 74,A 85.4316,B 24.8654,C -2.6773,E1 24.9952,E2 -1.4536} C_DIS
LIN {X 0.0559,Y 62.6502,Z 74,A 82.978,B 24.8652,C -2.6794,E1 25.0021,E2 0.9948} C_DIS
LIN {X 2.6146,Y 62.5948,Z 74,A 80.6779,B 24.8651,C -2.6805,E1 25.0085,E2 3.2918} C_DIS
LIN {X 5.2215,Y 62.4318,Z 74,A 78.5381,B 24.8645,C -2.6858,E1 25.0144,E2 5.4181} C_DIS
LIN {X 7.2631,Y 62.2269,Z 74,A 76.4394,B 24.8651,C -2.6807,E1 25.0203,E2 7.5274} C_DIS
LIN {X 9.7893,Y 61.8802,Z 74,A 74.0543,B 24.8652,C -2.6789,E1 25.0269,E2 9.9146} C_DIS
LIN {X 12.3027,Y 61.4303,Z 74,A 71.7118,B 24.8653,C -2.6778,E1 25.0333,E2 12.257} C_DIS
LIN {X 15.1473,Y 60.7914,Z 74,A 68.9696,B 24.8657,C -2.6747,E1 25.0407,E2 15.0027} C_DIS
LIN {X 17.8661,Y 60.0479,Z 74,A 65.6951,B 24.8674,C -2.6576,E1 25.0496,E2 18.3122} C_DIS
LIN {X 21.5742,Y 58.8176,Z 74,A 62.8659,B 24.866,C -2.671,E1 25.057,E2 21.1039} C_DIS
LIN {X 23.9782,Y 57.8803,Z 74,A 60.3676,B 24.8666,C -2.6655,E1 25.0635,E2 23.6096} C_DIS
LIN {X 26.6707,Y 56.6893,Z 74,A 57.7181,B 24.8668,C -2.6634,E1 25.0702,E2 26.2573} C_DIS
LIN {X 29.5952,Y 55.2192,Z 74,A 54.9097,B 24.8668,C -2.6638,E1 25.0771,E2 29.057} C_DIS
LIN {X 31.91,Y 53.9138,Z 74,A 52.545,B 24.8669,C -2.6619,E1 25.0828,E2 31.4191} C_DIS
LIN {X 35.283,Y 51.7696,Z 74,A 48.7763,B 24.8678,C -2.6536,E1 25.0917,E2 35.1951} C_DIS
LIN {X 37.5063,Y 50.1821,Z 74,A 46.3216,B 24.8681,C -2.6504,E1 25.0972,E2 37.6488} C_DIS
LIN {X 39.1529,Y 48.9094,Z 74,A 44.0252,B 24.8694,C -2.6377,E1 25.1023,E2 39.9666} C_DIS
LIN {X 43.2508,Y 45.3256,Z 74,A 39.5906,B 24.8691,C -2.6408,E1 25.1114,E2 44.3762} C_DIS
LIN {X 46.1649,Y 42.3526,Z 74,A 35.471,B 24.8706,C -2.6252,E1 25.1194,E2 48.5148} C_DIS
LIN {X 48.4349,Y 39.7384,Z 74,A 32.6002,B 24.8706,C -2.625,E1 25.1246,E2 51.373} C_DIS
LIN {X 50.3618,Y 37.2657,Z 74,A 29.7396,B 24.8713,C -2.6183,E1 25.1294,E2 54.2358} C_DIS
LIN {X 51.7535,Y 35.3067,Z 74,A 27.5303,B 24.8718,C -2.6126,E1 25.133,E2 56.4478} C_DIS
LIN {X 53.1855,Y 33.1097,Z 74,A 25.3884,B 24.8718,C -2.6127,E1 25.1362,E2 58.5787} C_DIS
LIN {X 54.392,Y 31.0881,Z 74,A 22.9093,B 24.8732,C -2.5991,E1 25.1397,E2 61.0772} C_DIS
LIN {X 55.5953,Y 28.883,Z 74,A 20.5937,B 24.8738,C -2.5925,E1 25.1427,E2 63.3963} C_DIS
LIN {X 56.9787,Y 26.0478,Z 74,A 17.7389,B 24.8745,C -2.5852,E1 25.1462,E2 66.253} C_DIS
LIN {X 58.4918,Y 22.4439,Z 74,A 14.2839,B 24.8752,C -2.578,E1 25.1498,E2 69.706} C_DIS
LIN {X 59.375,Y 19.9888,Z 74,A 11.9162,B 24.8759,C -2.5715,E1 25.152,E2 72.0758} C_DIS
LIN {X 60.2305,Y 17.2412,Z 74,A 9.3512,B 24.8765,C -2.5653,E1 25.154,E2 74.6407} C_DIS
LIN {X 60.8607,Y 14.8633,Z 74,A 7.1582,B 24.877,C -2.5599,E1 25.1555,E2 76.8337} C_DIS
LIN {X 61.3966,Y 12.4669,Z 74,A 4.7973,B 24.8779,C -2.5502,E1 25.1569,E2 79.2038} C_DIS
LIN {X 61.8791,Y 9.7964,Z 74,A 2.2205,B 24.8789,C -2.5402,E1 25.1581,E2 81.7892} C_DIS
LIN {X 62.2569,Y 7.0066,Z 74,A -0.1504,B 24.8792,C -2.5372,E1 25.1589,E2 84.1531} C_DIS
LIN {X 62.4774,Y 4.6516,Z 74,A -2.3422,B 24.8799,C -2.5297,E1 25.1595,E2 86.3497} C_DIS
LIN {X 62.6094,Y 2.2637,Z 74,A -4.2379,B 24.8799,C -2.5301,E1 25.1597,E2 88.2332} C_DIS
LIN {X 62.6484,Y 0.2343,Z 74,A -6.1677,B 24.8806,C -2.5224,E1 25.1597,E2 90.1696} C_DIS
LIN {X 62.6215,Y -1.8699,Z 74,A -8.4814,B 24.8821,C -2.5066,E1 25.1597,E2 92.5069} C_DIS
LIN {X 62.4297,Y -5.2486,Z 74,A -11.4425,B 24.8827,C -2.5001,E1 25.159,E2 95.4658} C_DIS
LIN {X 62.0865,Y -8.3858,Z 74,A -14.0803,B 24.883,C -2.4972,E1 25.1582,E2 98.095} C_DIS
LIN {X 61.7256,Y -10.725,Z 74,A -16.4107,B 24.884,C -2.4862,E1 25.1571,E2 100.4377} C_DIS
LIN {X 61.2077,Y -13.3624,Z 74,A -18.7278,B 24.8844,C -2.482,E1 25.1558,E2 102.7512} C_DIS
LIN {X 60.7914,Y -15.1472,Z 74,A -20.5022,B 24.8851,C -2.4743,E1 25.1546,E2 104.5335} C_DIS
LIN {X 60.0188,Y -17.9637,Z 74,A -23.1391,B 24.8858,C -2.4669,E1 25.1526,E2 107.1729} C_DIS
LIN {X 59.0347,Y -20.9719,Z 74,A -26.4597,B 24.8876,C -2.4475,E1 25.1496,E2 110.5206} C_DIS
LIN {X 57.9057,Y -23.9159,Z 74,A -29.631,B 24.889,C -2.4317,E1 25.1462,E2 113.7118} C_DIS
LIN {X 56.0425,Y -28.0039,Z 74,A -32.9685,B 24.8884,C -2.4385,E1 25.1422,E2 117.0151} C_DIS
LIN {X 54.9812,Y -30.0341,Z 74,A -35.155,B 24.8892,C -2.4302,E1 25.1393,E2 119.2098} C_DIS
LIN {X 53.5397,Y -32.5338,Z 74,A -37.5485,B 24.8892,C -2.4288,E1 25.1359,E2 121.5943} C_DIS
LIN {X 52.2483,Y -34.5697,Z 74,A -39.7417,B 24.8898,C -2.4229,E1 25.1326,E2 123.7904} C_DIS
LIN {X 50.9121,Y -36.5092,Z 74,A -41.8625,B 24.8903,C -2.4179,E1 25.1292,E2 125.9128} C_DIS
LIN {X 49.0909,Y -38.9234,Z 74,A -44.7346,B 24.8912,C -2.408,E1 25.1243,E2 128.7947} C_DIS
LIN {X 47.2628,Y -41.124,Z 74,A -47.2895,B 24.8917,C -2.4028,E1 25.1197,E2 131.3502} C_DIS
LIN {X 45.3532,Y -43.2221,Z 74,A -49.6376,B 24.8917,C -2.4023,E1 25.1152,E2 133.6891} C_DIS
LIN {X 43.7821,Y -44.8129,Z 74,A -52.2511,B 24.8934,C -2.3837,E1 25.11,E2 136.3356} C_DIS
LIN {X 41.2315,Y -47.1689,Z 74,A -55.1949,B 24.8935,C -2.382,E1 25.1039,E2 139.2717} C_DIS
LIN {X 38.843,Y -49.1545,Z 74,A -57.5257,B 24.893,C -2.3881,E1 25.0989,E2 141.5792} C_DIS
LIN {X 36.4792,Y -50.9333,Z 74,A -60.7478,B 24.8946,C -2.3701,E1 25.0916,E2 144.8323} C_DIS
LIN {X 34.048,Y -52.5903,Z 74,A -63.2539,B 24.8946,C -2.3693,E1 25.0858,E2 147.3321} C_DIS
LIN {X 31.9904,Y -53.8663,Z 74,A -65.4194,B 24.8949,C -2.3664,E1 25.0806,E2 149.4977} C_DIS
LIN {X 30.4567,Y -54.748,Z 74,A -67.3378,B 24.8958,C -2.3565,E1 25.0759,E2 151.4339} C_DIS
LIN {X 27.5154,Y -56.2847,Z 74,A -69.8751,B 24.8952,C -2.3631,E1 25.0697,E2 153.9484} C_DIS
LIN {X 24.5812,Y -57.6262,Z 74,A -73.7163,B 24.8974,C -2.3381,E1 25.0597,E2 157.8396} C_DIS
LIN {X 20.6955,Y -59.1324,Z 74,A -76.5281,B 24.8958,C -2.3561,E1 25.0525,E2 160.6026} C_DIS
LIN {X 17.734,Y -60.0871,Z 74,A -79.6355,B 24.8967,C -2.3467,E1 25.0442,E2 163.7266} C_DIS
LIN {X 15.3937,Y -60.7291,Z 74,A -81.9274,B 24.897,C -2.3428,E1 25.038,E2 166.0243} C_DIS
LIN {X 12.8592,Y -61.316,Z 74,A -84.3485,B 24.8973,C -2.3397,E1 25.0314,E2 168.4496} C_DIS
LIN {X 9.6188,Y -61.9066,Z 74,A -87.2354,B 24.8973,C -2.3402,E1 25.0234,E2 171.3322} C_DIS
LIN {X 7.307,Y -62.2218,Z 74,A -89.3139,B 24.8973,C -2.3402,E1 25.0177,E2 173.4092} C_DIS
LIN {X 4.4829,Y -62.4893,Z 74,A -91.9887,B 24.8975,C -2.337,E1 25.0102,E2 176.0899} C_DIS
Enddeposition()
END
